C01821=1016.661,-35.852,383.395,-24.107,21.573,-43.343
C01822=1016.661,-36.185,383.421,-24.107,21.574,-43.347
C01823=1016.662,-36.517,383.447,-24.106,21.574,-43.352
C01824=1016.663,-36.850,383.473,-24.105,21.574,-43.357
C01825=1016.662,-37.183,383.498,-24.105,21.575,-43.361
C01826=1016.663,-37.515,383.525,-24.104,21.575,-43.366
C01827=1016.663,-37.848,383.550,-24.103,21.576,-43.371
C01828=1016.663,-38.180,383.576,-24.102,21.576,-43.376
C01829=1016.664,-38.513,383.602,-24.102,21.577,-43.380
C01830=1016.664,-38.846,383.627,-24.101,21.577,-43.385
C01831=1016.665,-39.178,383.654,-24.101,21.578,-43.389
C01832=1016.664,-39.511,383.679,-24.100,21.578,-43.394
C01833=1016.665,-39.844,383.705,-24.100,21.579,-43.398
C01834=1016.664,-40.177,383.731,-24.099,21.579,-43.404
C01835=1016.665,-40.509,383.757,-24.098,21.580,-43.409
C01836=1016.665,-40.842,383.782,-24.098,21.580,-43.413
C01837=1016.665,-41.174,383.808,-24.097,21.580,-43.418
C01838=1016.665,-41.507,383.834,-24.096,21.582,-43.422
C01839=1016.665,-41.839,383.859,-24.096,21.582,-43.427
C01840=1016.666,-42.172,383.885,-24.095,21.582,-43.431
C01841=1016.666,-42.504,383.911,-24.094,21.583,-43.437
C01842=1016.666,-42.837,383.936,-24.094,21.583,-43.442
C01843=1016.665,-43.169,383.962,-24.093,21.583,-43.446
C01844=1016.666,-43.502,383.987,-24.092,21.584,-43.451
C01845=1016.665,-43.835,384.013,-24.092,21.585,-43.455
C01846=1016.665,-44.167,384.039,-24.091,21.585,-43.461
C01847=1016.665,-44.500,384.064,-24.091,21.586,-43.465
C01848=1016.666,-44.833,384.090,-24.090,21.586,-43.470
C01849=1016.666,-45.165,384.116,-24.089,21.586,-43.475
C01850=1016.666,-45.498,384.141,-24.089,21.587,-43.479
C01851=1016.665,-45.830,384.167,-24.088,21.588,-43.485
C01852=1016.665,-46.162,384.192,-24.088,21.588,-43.488
C01853=1016.665,-46.495,384.217,-24.087,21.588,-43.494
C01854=1016.665,-46.827,384.243,-24.086,21.590,-43.498
C01855=1016.664,-47.160,384.269,-24.086,21.589,-43.503
C01856=1016.664,-47.493,384.294,-24.085,21.589,-43.508
C01857=1016.664,-47.825,384.320,-24.084,21.591,-43.512
C01858=1016.664,-48.158,384.345,-24.083,21.591,-43.518
C01859=1016.664,-48.490,384.370,-24.083,21.592,-43.522
C01860=1016.664,-48.822,384.396,-24.082,21.592,-43.527
C01861=1016.664,-49.155,384.421,-24.081,21.592,-43.532
C01862=1016.664,-49.487,384.447,-24.081,21.593,-43.536
C01863=1016.663,-49.820,384.472,-24.080,21.593,-43.542
C01864=1016.663,-50.152,384.497,-24.080,21.595,-43.546
C01865=1016.662,-50.484,384.522,-24.079,21.594,-43.551
C01866=1016.662,-50.817,384.548,-24.079,21.595,-43.555
C01867=1016.662,-51.149,384.573,-24.078,21.596,-43.560
C01868=1016.661,-51.482,384.599,-24.077,21.596,-43.566
C01869=1016.660,-51.814,384.624,-24.077,21.597,-43.570
C01870=1016.661,-52.147,384.649,-24.076,21.597,-43.575
C01871=1016.660,-52.479,384.674,-24.075,21.597,-43.579
C01872=1016.659,-52.811,384.700,-24.075,21.598,-43.584
C01873=1016.659,-53.144,384.725,-24.074,21.598,-43.589
C01874=1016.658,-53.476,384.750,-24.074,21.600,-43.594
C01875=1016.658,-53.808,384.776,-24.073,21.599,-43.599
C01876=1016.658,-54.140,384.800,-24.072,21.600,-43.603
C01877=1016.657,-54.473,384.826,-24.072,21.601,-43.608
C01878=1016.656,-54.805,384.851,-24.071,21.601,-43.613
C01879=1016.656,-55.137,384.876,-24.070,21.602,-43.618
C01880=1016.655,-55.469,384.901,-24.070,21.602,-43.623
C01881=1016.655,-55.803,384.926,-24.069,21.603,-43.627
C01882=1016.655,-56.136,384.951,-24.068,21.603,-43.632
C01883=1016.653,-56.468,384.977,-24.068,21.603,-43.637
C01884=1016.654,-56.801,385.002,-24.067,21.605,-43.642
C01885=1016.653,-57.135,385.027,-24.066,21.604,-43.647
C01886=1016.652,-57.468,385.052,-24.066,21.605,-43.652
C01887=1016.651,-57.803,385.077,-24.065,21.606,-43.656
C01888=1016.650,-58.136,385.102,-24.064,21.606,-43.662
C01889=1016.650,-58.471,385.128,-24.064,21.607,-43.666
C01890=1016.650,-58.806,385.153,-24.063,21.607,-43.671
C01891=1016.649,-59.141,385.178,-24.062,21.608,-43.676
C01892=1016.647,-59.477,385.203,-24.062,21.608,-43.680
C01893=1016.647,-59.813,385.228,-24.061,21.609,-43.686
C01894=1016.646,-60.149,385.254,-24.060,21.609,-43.691
C01895=1016.645,-60.486,385.280,-24.060,21.610,-43.695
C01896=1016.645,-60.823,385.304,-24.059,21.610,-43.700
C01897=1016.644,-61.162,385.330,-24.059,21.611,-43.706
C01898=1016.643,-61.499,385.355,-24.058,21.611,-43.710
C01899=1016.642,-61.838,385.381,-24.057,21.612,-43.715
C01900=1016.641,-62.177,385.406,-24.057,21.612,-43.720
C01901=1016.640,-62.515,385.432,-24.056,21.614,-43.725
C01902=1016.640,-62.855,385.457,-24.055,21.613,-43.730
C01903=1016.638,-63.195,385.482,-24.055,21.614,-43.735
C01904=1016.637,-63.535,385.507,-24.054,21.615,-43.739
C01905=1016.636,-63.876,385.533,-24.053,21.616,-43.745
C01906=1016.636,-64.217,385.558,-24.053,21.615,-43.750
C01907=1016.634,-64.558,385.584,-24.052,21.617,-43.754
C01908=1016.634,-64.900,385.609,-24.051,21.617,-43.759
C01909=1016.632,-65.242,385.635,-24.051,21.618,-43.765
C01910=1016.631,-65.584,385.660,-24.050,21.617,-43.770
C01911=1016.630,-65.926,385.686,-24.050,21.619,-43.774
C01912=1016.629,-66.269,385.711,-24.049,21.619,-43.780
C01913=1016.628,-66.612,385.737,-24.048,21.620,-43.785
C01914=1016.626,-66.955,385.762,-24.048,21.620,-43.789
C01915=1016.626,-67.298,385.787,-24.047,21.621,-43.795
C01916=1016.624,-67.641,385.814,-24.046,21.621,-43.800
C01917=1016.623,-67.984,385.839,-24.045,21.622,-43.805
C01918=1016.621,-68.328,385.864,-24.045,21.622,-43.809
C01919=1016.620,-68.672,385.890,-24.044,21.623,-43.815
C01920=1016.620,-69.016,385.915,-24.043,21.623,-43.820
C01921=1016.619,-69.360,385.941,-24.043,21.624,-43.824
C01922=1016.617,-69.704,385.966,-24.042,21.624,-43.829
C01923=1016.615,-70.047,385.992,-24.041,21.625,-43.835
C01924=1016.614,-70.391,386.017,-24.041,21.625,-43.840
C01925=1016.613,-70.736,386.042,-24.040,21.626,-43.844
C01926=1016.611,-71.080,386.068,-24.040,21.627,-43.850
C01927=1016.610,-71.424,386.093,-24.039,21.627,-43.855
C01928=1016.609,-71.768,386.118,-24.038,21.628,-43.861
C01929=1016.608,-72.112,386.144,-24.038,21.628,-43.865
C01930=1016.606,-72.456,386.169,-24.037,21.629,-43.870
C01931=1016.604,-72.800,386.195,-24.036,21.629,-43.875
C01932=1016.603,-73.144,386.220,-24.035,21.630,-43.881
C01933=1016.602,-73.488,386.245,-24.035,21.630,-43.885
C01934=1016.600,-73.831,386.270,-24.034,21.631,-43.890
C01935=1016.598,-74.175,386.296,-24.033,21.632,-43.896
C01936=1016.596,-74.519,386.321,-24.033,21.632,-43.901
C01937=1016.595,-74.862,386.346,-24.032,21.633,-43.905
C01938=1016.594,-75.206,386.372,-24.031,21.633,-43.911
C01939=1016.592,-75.549,386.397,-24.031,21.634,-43.916
C01940=1016.590,-75.892,386.422,-24.030,21.634,-43.920
C01941=1016.589,-76.235,386.447,-24.030,21.635,-43.926
C01942=1016.587,-76.578,386.472,-24.029,21.635,-43.931
C01943=1016.585,-76.920,386.498,-24.028,21.636,-43.936
C01944=1016.583,-77.263,386.522,-24.028,21.636,-43.940
C01945=1016.582,-77.604,386.547,-24.027,21.637,-43.946
C01946=1016.580,-77.946,386.572,-24.026,21.637,-43.951
C01947=1016.579,-78.288,386.597,-24.026,21.639,-43.955
C01948=1016.577,-78.629,386.622,-24.025,21.638,-43.960
C01949=1016.575,-78.970,386.647,-24.024,21.639,-43.966
C01950=1016.573,-79.310,386.672,-24.023,21.639,-43.971
C01951=1016.571,-79.651,386.697,-24.023,21.641,-43.975
C01952=1016.570,-79.990,386.722,-24.022,21.641,-43.981
C01953=1016.568,-80.329,386.746,-24.021,21.641,-43.986
C01954=1016.566,-80.669,386.770,-24.021,21.643,-43.990
C01955=1016.564,-81.007,386.796,-24.020,21.643,-43.995
C01956=1016.562,-81.345,386.820,-24.020,21.643,-44.001
C01957=1016.560,-81.683,386.844,-24.019,21.644,-44.005
C01958=1016.558,-82.020,386.869,-24.018,21.645,-44.010
C01959=1016.556,-82.358,386.894,-24.018,21.645,-44.016
C01960=1016.555,-82.694,386.918,-24.017,21.645,-44.021
C01961=1016.552,-83.030,386.942,-24.016,21.646,-44.025
C01962=1016.550,-83.366,386.967,-24.016,21.647,-44.031
C01963=1016.549,-83.701,386.991,-24.015,21.647,-44.036
C01964=1016.547,-84.036,387.015,-24.015,21.648,-44.040
C01965=1016.544,-84.370,387.039,-24.014,21.648,-44.045
C01966=1016.542,-84.719,387.065,-24.013,21.649,-44.051
C01967=1016.540,-85.117,387.094,-24.012,21.650,-44.056
C01968=1016.538,-85.330,387.109,-24.012,21.649,-44.060
C01969=1016.538,-85.543,387.124,-24.012,21.649,-44.062
C01970=1016.535,-85.951,387.154,-24.011,21.650,-44.067
C01971=1016.532,-86.311,387.179,-24.010,21.651,-44.073
C01972=1016.531,-86.640,387.203,-24.009,21.652,-44.078
C01973=1016.528,-86.963,387.226,-24.009,21.652,-44.082
C01974=1016.526,-87.279,387.250,-24.008,21.653,-44.088
C01975=1016.524,-87.591,387.272,-24.007,21.653,-44.093
C01976=1016.522,-87.902,387.294,-24.007,21.654,-44.097
C01977=1016.520,-88.215,387.317,-24.006,21.654,-44.102
C01978=1016.518,-88.533,387.340,-24.006,21.655,-44.106
C01979=1016.515,-88.905,387.367,-24.005,21.656,-44.114
C01980=1016.514,-89.123,387.382,-24.004,21.656,-44.117
C01981=1016.512,-89.358,387.399,-24.004,21.656,-44.119
C01982=1016.510,-89.596,387.416,-24.004,21.656,-44.121
C01983=1016.509,-89.827,387.433,-24.004,21.657,-44.123
C01984=1016.506,-90.233,387.462,-24.003,21.658,-44.130
C01985=1016.503,-90.571,387.486,-24.002,21.658,-44.136
C01986=1016.502,-90.901,387.510,-24.001,21.659,-44.141
C01987=1016.499,-91.230,387.533,-24.001,21.660,-44.145
C01988=1016.496,-91.558,387.557,-24.000,21.660,-44.150
C01989=1016.494,-91.887,387.580,-23.999,21.660,-44.156
C01990=1016.492,-92.215,387.604,-23.999,21.661,-44.160
C01991=1016.489,-92.542,387.627,-23.998,21.662,-44.165
C01992=1016.487,-92.868,387.651,-23.998,21.662,-44.169
C01993=1016.484,-93.195,387.673,-23.997,21.663,-44.175
C01994=1016.482,-93.520,387.697,-23.996,21.663,-44.180
C01995=1016.479,-93.846,387.721,-23.996,21.664,-44.184
C01996=1016.477,-94.171,387.743,-23.995,21.664,-44.189
C01997=1016.474,-94.494,387.766,-23.994,21.665,-44.193
C01998=1016.471,-94.818,387.790,-23.994,21.666,-44.199
C01999=1016.469,-95.140,387.812,-23.993,21.666,-44.204
C02000=1016.467,-95.463,387.836,-23.993,21.666,-44.207
C02001=1016.465,-95.786,387.859,-23.992,21.667,-44.213
C02002=1016.461,-96.108,387.882,-23.991,21.668,-44.217
C02003=1016.459,-96.429,387.904,-23.991,21.668,-44.222
C02004=1016.456,-96.751,387.927,-23.990,21.669,-44.226
C02005=1016.453,-97.072,387.950,-23.989,21.669,-44.231
C02006=1016.451,-97.393,387.973,-23.989,21.670,-44.236
C02007=1016.449,-97.713,387.995,-23.988,21.670,-44.241
C02008=1016.446,-98.035,388.019,-23.987,21.670,-44.246
C02009=1016.443,-98.356,388.041,-23.987,21.672,-44.250
C02010=1016.441,-98.676,388.064,-23.986,21.671,-44.255
C02011=1016.438,-98.998,388.087,-23.986,21.673,-44.260
C02012=1016.436,-99.319,388.109,-23.985,21.673,-44.265
C02013=1016.432,-99.640,388.132,-23.985,21.673,-44.268
C02014=1016.429,-99.962,388.154,-23.984,21.674,-44.274
C02015=1016.427,-100.284,388.177,-23.983,21.675,-44.278
C02016=1016.424,-100.606,388.200,-23.983,21.675,-44.283
C02017=1016.421,-100.928,388.223,-23.982,21.676,-44.287
C02018=1016.419,-101.252,388.246,-23.981,21.676,-44.292
C02019=1016.415,-101.575,388.269,-23.981,21.677,-44.298
C02020=1016.412,-101.899,388.292,-23.980,21.677,-44.302
C02021=1016.409,-102.224,388.315,-23.980,21.678,-44.307
C02022=1016.407,-102.549,388.337,-23.979,21.679,-44.311
C02023=1016.403,-102.874,388.360,-23.978,21.679,-44.316
C02024=1016.400,-103.201,388.384,-23.978,21.680,-44.320
C02025=1016.397,-103.527,388.406,-23.977,21.680,-44.326
C02026=1016.395,-103.854,388.429,-23.976,21.681,-44.331
C02027=1016.392,-104.181,388.452,-23.976,21.681,-44.335
C02028=1016.388,-104.509,388.475,-23.975,21.681,-44.340
C02029=1016.385,-104.837,388.498,-23.975,21.683,-44.344
C02030=1016.381,-105.165,388.521,-23.974,21.683,-44.350
C02031=1016.379,-105.494,388.545,-23.974,21.684,-44.354
C02032=1016.376,-105.823,388.567,-23.973,21.684,-44.359
C02033=1016.372,-106.151,388.591,-23.972,21.685,-44.365
C02034=1016.369,-106.480,388.614,-23.972,21.685,-44.368
C02035=1016.365,-106.809,388.637,-23.971,21.685,-44.374
C02036=1016.363,-107.139,388.661,-23.971,21.687,-44.378
C02037=1016.359,-107.467,388.683,-23.970,21.687,-44.383
C02038=1016.356,-107.797,388.706,-23.969,21.687,-44.388
C02039=1016.353,-108.125,388.729,-23.969,21.688,-44.392
C02040=1016.349,-108.455,388.752,-23.968,21.689,-44.398
C02041=1016.346,-108.784,388.775,-23.967,21.689,-44.402
C02042=1016.343,-109.112,388.798,-23.967,21.689,-44.407
C02043=1016.339,-109.442,388.821,-23.966,21.690,-44.412
C02044=1016.336,-109.770,388.844,-23.965,21.691,-44.416
C02045=1016.332,-110.100,388.867,-23.965,21.691,-44.422
C02046=1016.329,-110.428,388.889,-23.964,21.692,-44.426
C02047=1016.325,-110.757,388.913,-23.963,21.692,-44.431
C02048=1016.322,-111.086,388.936,-23.963,21.693,-44.436
C02049=1016.318,-111.414,388.958,-23.962,21.693,-44.440
C02050=1016.314,-111.744,388.981,-23.962,21.694,-44.446
C02051=1016.311,-112.072,389.004,-23.961,21.695,-44.449
C02052=1016.308,-112.401,389.027,-23.960,21.695,-44.455
C02053=1016.304,-112.730,389.050,-23.960,21.696,-44.459
C02054=1016.300,-113.058,389.073,-23.959,21.696,-44.464
C02055=1016.297,-113.387,389.096,-23.958,21.697,-44.470
C02056=1016.293,-113.716,389.119,-23.958,21.697,-44.473
C02057=1016.289,-114.044,389.141,-23.957,21.698,-44.479
C02058=1016.285,-114.373,389.165,-23.957,21.699,-44.483
C02059=1016.282,-114.701,389.187,-23.956,21.699,-44.488
C02060=1016.278,-115.031,389.210,-23.956,21.700,-44.492
C02061=1016.274,-115.359,389.232,-23.955,21.700,-44.497
C02062=1016.270,-115.688,389.256,-23.954,21.701,-44.503
C02063=1016.267,-116.016,389.278,-23.954,21.701,-44.507
C02064=1016.263,-116.345,389.301,-23.953,21.701,-44.512
C02065=1016.259,-116.673,389.324,-23.953,21.703,-44.516
C02066=1016.255,-117.001,389.346,-23.952,21.703,-44.521
C02067=1016.251,-117.330,389.369,-23.951,21.704,-44.525
C02068=1016.248,-117.659,389.391,-23.951,21.704,-44.531
C02069=1016.243,-117.987,389.414,-23.950,21.705,-44.535
C02070=1016.240,-118.315,389.437,-23.949,21.705,-44.540
C02071=1016.236,-118.644,389.459,-23.949,21.705,-44.545
C02072=1016.231,-118.972,389.482,-23.948,21.707,-44.549
C02073=1016.227,-119.301,389.505,-23.948,21.707,-44.554
C02074=1016.224,-119.629,389.528,-23.947,21.707,-44.558
C02075=1016.219,-119.958,389.550,-23.946,21.708,-44.564
C02076=1016.216,-120.286,389.573,-23.946,21.709,-44.568
C02077=1016.212,-120.614,389.595,-23.945,21.709,-44.573
C02078=1016.207,-120.943,389.618,-23.945,21.710,-44.577
C02079=1016.203,-121.270,389.641,-23.944,21.710,-44.582
C02080=1016.199,-121.599,389.663,-23.944,21.711,-44.586
C02081=1016.195,-121.928,389.685,-23.943,21.711,-44.591
C02082=1016.190,-122.256,389.708,-23.942,21.712,-44.597
C02083=1016.186,-122.584,389.730,-23.942,21.713,-44.601
C02084=1016.182,-122.913,389.754,-23.941,21.713,-44.606
C02085=1016.178,-123.241,389.776,-23.940,21.714,-44.610
C02086=1016.173,-123.569,389.799,-23.940,21.714,-44.615
C02087=1016.169,-123.897,389.820,-23.939,21.715,-44.620
C02088=1016.165,-124.225,389.843,-23.939,21.715,-44.625
C02089=1016.160,-124.554,389.866,-23.938,21.716,-44.628
C02090=1016.157,-124.882,389.888,-23.937,21.717,-44.634
C02091=1016.152,-125.210,389.911,-23.937,21.717,-44.638
C02092=1016.147,-125.538,389.933,-23.936,21.717,-44.643
C02093=1016.143,-125.867,389.956,-23.936,21.719,-44.647
C02094=1016.139,-126.195,389.978,-23.935,21.719,-44.652
C02095=1016.134,-126.523,390.000,-23.935,21.720,-44.657
C02096=1016.129,-126.850,390.023,-23.934,21.720,-44.662
C02097=1016.125,-127.179,390.046,-23.933,21.720,-44.667
C02098=1016.120,-127.507,390.068,-23.933,21.721,-44.671
C02099=1016.116,-127.836,390.090,-23.932,21.721,-44.676
C02100=1016.111,-128.163,390.113,-23.931,21.722,-44.680
C02101=1016.107,-128.492,390.135,-23.931,21.723,-44.686
C02102=1016.102,-128.819,390.157,-23.930,21.723,-44.689
C02103=1016.097,-129.148,390.180,-23.929,21.723,-44.695
C02104=1016.093,-129.476,390.202,-23.929,21.725,-44.699
C02105=1016.088,-129.804,390.224,-23.928,21.724,-44.704
C02106=1016.083,-130.132,390.247,-23.928,21.726,-44.708
C02107=1016.078,-130.460,390.269,-23.927,21.726,-44.713
C02108=1016.074,-130.789,390.292,-23.927,21.726,-44.717
C02109=1016.069,-131.116,390.314,-23.926,21.727,-44.723
C02110=1016.064,-131.445,390.336,-23.926,21.728,-44.726
C02111=1016.059,-131.772,390.358,-23.925,21.728,-44.732
C02112=1016.054,-132.100,390.381,-23.924,21.729,-44.736
C02113=1016.050,-132.428,390.403,-23.924,21.729,-44.741
C02114=1016.044,-132.756,390.425,-23.923,21.730,-44.745
C02115=1016.039,-133.085,390.447,-23.922,21.731,-44.750
C02116=1016.034,-133.412,390.469,-23.922,21.731,-44.754
C02117=1016.029,-133.740,390.492,-23.921,21.731,-44.759
C02118=1016.025,-134.069,390.514,-23.921,21.732,-44.763
C02119=1016.426,-134.039,390.264,-23.921,21.732,-44.763
C02120=1016.431,-133.712,390.241,-23.921,21.731,-44.759
C02121=1016.436,-133.383,390.220,-23.922,21.731,-44.754
C02122=1016.441,-133.056,390.197,-23.922,21.731,-44.750
C02123=1016.446,-132.727,390.175,-23.923,21.730,-44.745
C02124=1016.450,-132.400,390.153,-23.924,21.729,-44.741
C02125=1016.455,-132.072,390.131,-23.924,21.729,-44.736
C02126=1016.460,-131.744,390.109,-23.925,21.728,-44.732
C02127=1016.464,-131.415,390.086,-23.926,21.728,-44.726
C02128=1016.469,-131.087,390.064,-23.926,21.727,-44.723
C02129=1016.474,-130.759,390.042,-23.927,21.726,-44.717
C02130=1016.477,-130.431,390.020,-23.927,21.726,-44.713
C02131=1016.483,-130.103,389.998,-23.928,21.726,-44.708
C02132=1016.487,-129.775,389.976,-23.928,21.724,-44.704
C02133=1016.492,-129.447,389.953,-23.929,21.725,-44.699
C02134=1016.496,-129.119,389.931,-23.929,21.723,-44.695
C02135=1016.501,-128.791,389.909,-23.930,21.723,-44.689
C02136=1016.505,-128.462,389.886,-23.931,21.723,-44.686
C02137=1016.510,-128.135,389.864,-23.931,21.722,-44.680
C02138=1016.514,-127.807,389.842,-23.932,21.721,-44.676
C02139=1016.519,-127.478,389.820,-23.933,21.721,-44.671
C02140=1016.523,-127.150,389.797,-23.933,21.720,-44.667
C02141=1016.527,-126.822,389.775,-23.934,21.720,-44.662
C02142=1016.532,-126.494,389.752,-23.935,21.720,-44.657
C02143=1016.536,-126.166,389.730,-23.935,21.719,-44.652
C02144=1016.540,-125.837,389.708,-23.936,21.719,-44.647
C02145=1016.545,-125.510,389.686,-23.936,21.717,-44.643
C02146=1016.549,-125.181,389.664,-23.937,21.717,-44.638
C02147=1016.553,-124.853,389.640,-23.937,21.717,-44.634
C02148=1016.557,-124.525,389.618,-23.938,21.716,-44.628
C02149=1016.561,-124.197,389.596,-23.939,21.715,-44.625
C02150=1016.566,-123.868,389.573,-23.939,21.715,-44.620
C02151=1016.569,-123.540,389.551,-23.940,21.714,-44.615
C02152=1016.574,-123.212,389.529,-23.940,21.714,-44.610
C02153=1016.579,-122.884,389.506,-23.941,21.713,-44.606
C02154=1016.582,-122.555,389.484,-23.942,21.713,-44.601
C02155=1016.586,-122.227,389.462,-23.942,21.712,-44.597
C02156=1016.591,-121.899,389.439,-23.943,21.711,-44.591
C02157=1016.595,-121.571,389.417,-23.944,21.711,-44.586
C02158=1016.598,-121.242,389.395,-23.944,21.710,-44.582
C02159=1016.602,-120.914,389.371,-23.945,21.710,-44.577
C02160=1016.606,-120.585,389.349,-23.945,21.709,-44.573
C02161=1016.610,-120.257,389.327,-23.946,21.709,-44.568
C02162=1016.615,-119.929,389.303,-23.946,21.708,-44.564
C02163=1016.618,-119.601,389.281,-23.947,21.707,-44.558
C02164=1016.622,-119.272,389.259,-23.948,21.707,-44.554
C02165=1016.626,-118.943,389.236,-23.948,21.707,-44.549
C02166=1016.630,-118.615,389.213,-23.949,21.705,-44.545
C02167=1016.634,-118.287,389.191,-23.949,21.705,-44.540
C02168=1016.638,-117.958,389.169,-23.950,21.705,-44.535
C02169=1016.641,-117.630,389.146,-23.951,21.704,-44.531
C02170=1016.645,-117.302,389.123,-23.951,21.704,-44.525
C02171=1016.649,-116.973,389.100,-23.952,21.703,-44.521
C02172=1016.652,-116.644,389.078,-23.953,21.703,-44.516
C02173=1016.656,-116.316,389.056,-23.953,21.701,-44.512
C02174=1016.660,-115.987,389.033,-23.954,21.701,-44.507
C02175=1016.664,-115.659,389.010,-23.954,21.701,-44.503
C02176=1016.667,-115.331,388.987,-23.955,21.700,-44.497
C02177=1016.671,-115.001,388.964,-23.956,21.700,-44.492
C02178=1016.674,-114.673,388.942,-23.956,21.699,-44.488
C02179=1016.677,-114.345,388.920,-23.957,21.699,-44.483
C02180=1016.682,-114.016,388.896,-23.957,21.698,-44.479
C02181=1016.685,-113.688,388.874,-23.958,21.697,-44.473
C02182=1016.689,-113.358,388.851,-23.958,21.697,-44.470
C02183=1016.693,-113.030,388.829,-23.959,21.696,-44.464
C02184=1016.696,-112.702,388.806,-23.960,21.696,-44.459
C02185=1016.699,-112.372,388.783,-23.960,21.695,-44.455
C02186=1016.702,-112.044,388.760,-23.961,21.695,-44.449
C02187=1016.707,-111.715,388.738,-23.962,21.694,-44.446
C02188=1016.710,-111.386,388.715,-23.962,21.693,-44.440
C02189=1016.713,-111.058,388.692,-23.963,21.693,-44.436
C02190=1016.717,-110.729,388.668,-23.963,21.692,-44.431
C02191=1016.720,-110.400,388.646,-23.964,21.692,-44.426
C02192=1016.723,-110.071,388.623,-23.965,21.691,-44.422
C02193=1016.726,-109.743,388.600,-23.965,21.691,-44.416
C02194=1016.730,-109.413,388.577,-23.966,21.690,-44.412
C02195=1016.733,-109.085,388.554,-23.967,21.689,-44.407
C02196=1016.737,-108.755,388.531,-23.967,21.689,-44.402
C02197=1016.740,-108.427,388.508,-23.968,21.689,-44.398
C02198=1016.743,-108.098,388.485,-23.969,21.688,-44.392
C02199=1016.746,-107.769,388.463,-23.969,21.687,-44.388
C02200=1016.749,-107.439,388.439,-23.970,21.687,-44.383
C02201=1016.752,-107.110,388.417,-23.971,21.687,-44.378
C02202=1016.756,-106.781,388.394,-23.971,21.685,-44.374
C02203=1016.759,-106.452,388.371,-23.972,21.685,-44.368
C02204=1016.762,-106.123,388.348,-23.972,21.685,-44.365
C02205=1016.765,-105.794,388.325,-23.973,21.684,-44.359
C02206=1016.768,-105.466,388.302,-23.974,21.684,-44.354
C02207=1016.771,-105.138,388.279,-23.974,21.683,-44.350
C02208=1016.774,-104.809,388.256,-23.975,21.683,-44.344
C02209=1016.777,-104.481,388.233,-23.975,21.681,-44.340
C02210=1016.780,-104.153,388.210,-23.976,21.681,-44.335
C02211=1016.783,-103.825,388.187,-23.976,21.681,-44.331
C02212=1016.786,-103.499,388.163,-23.977,21.680,-44.326
C02213=1016.789,-103.173,388.141,-23.978,21.680,-44.320
C02214=1016.791,-102.847,388.118,-23.978,21.679,-44.316
C02215=1016.795,-102.521,388.095,-23.979,21.679,-44.311
C02216=1016.798,-102.196,388.072,-23.980,21.678,-44.307
C02217=1016.800,-101.871,388.050,-23.980,21.677,-44.302
C02218=1016.803,-101.546,388.027,-23.981,21.677,-44.298
C02219=1016.806,-101.223,388.004,-23.981,21.676,-44.292
C02220=1016.809,-100.900,387.981,-23.982,21.676,-44.287
C02221=1016.812,-100.577,387.959,-23.983,21.675,-44.283
C02222=1016.815,-100.255,387.936,-23.983,21.675,-44.278
C02223=1016.817,-99.933,387.913,-23.984,21.674,-44.274
C02224=1016.820,-99.612,387.890,-23.985,21.673,-44.268
C02225=1016.822,-99.291,387.868,-23.985,21.673,-44.265
C02226=1016.826,-98.970,387.845,-23.986,21.673,-44.260
C02227=1016.828,-98.649,387.823,-23.986,21.671,-44.255
C02228=1016.831,-98.327,387.800,-23.987,21.672,-44.250
C02229=1016.833,-98.007,387.777,-23.987,21.670,-44.246
C02230=1016.836,-97.686,387.755,-23.988,21.670,-44.241
C02231=1016.838,-97.365,387.732,-23.989,21.670,-44.236
C02232=1016.841,-97.044,387.708,-23.989,21.669,-44.231
C02233=1016.843,-96.723,387.686,-23.990,21.669,-44.226
C02234=1016.846,-96.402,387.663,-23.991,21.668,-44.222
C02235=1016.849,-96.080,387.640,-23.991,21.668,-44.217
C02236=1016.851,-95.757,387.617,-23.992,21.667,-44.213
C02237=1016.854,-95.436,387.595,-23.993,21.666,-44.207
C02238=1016.856,-95.113,387.572,-23.993,21.666,-44.204
C02239=1016.858,-94.790,387.549,-23.994,21.666,-44.199
C02240=1016.861,-94.466,387.526,-23.994,21.665,-44.193
C02241=1016.863,-94.142,387.503,-23.995,21.664,-44.189
C02242=1016.866,-93.818,387.479,-23.996,21.664,-44.184
C02243=1016.868,-93.493,387.457,-23.996,21.663,-44.180
C02244=1016.871,-93.167,387.433,-23.997,21.663,-44.175
C02245=1016.873,-92.841,387.410,-23.998,21.662,-44.169
C02246=1016.875,-92.513,387.386,-23.998,21.662,-44.165
C02247=1016.878,-92.186,387.363,-23.999,21.661,-44.160
C02248=1016.880,-91.859,387.340,-23.999,21.660,-44.156
C02249=1016.882,-91.530,387.316,-24.000,21.660,-44.150
C02250=1016.885,-91.201,387.292,-24.001,21.660,-44.145
C02251=1016.887,-90.873,387.269,-24.001,21.659,-44.141
C02252=1016.889,-90.543,387.246,-24.002,21.658,-44.136
C02253=1016.891,-90.205,387.222,-24.003,21.658,-44.130
C02254=1016.894,-89.799,387.193,-24.004,21.657,-44.123
C02255=1016.896,-89.568,387.176,-24.004,21.656,-44.121
C02256=1016.898,-89.330,387.159,-24.004,21.656,-44.119
C02257=1016.899,-89.096,387.142,-24.004,21.656,-44.117
C02258=1016.901,-88.877,387.126,-24.005,21.656,-44.114
C02259=1016.903,-88.506,387.100,-24.006,21.655,-44.106
C02260=1016.905,-88.187,387.077,-24.006,21.654,-44.102
C02261=1016.907,-87.874,387.054,-24.007,21.654,-44.097
C02262=1016.908,-87.564,387.032,-24.007,21.653,-44.093
C02263=1016.911,-87.251,387.009,-24.008,21.653,-44.088
C02264=1016.913,-86.935,386.987,-24.009,21.652,-44.082
C02265=1016.915,-86.612,386.964,-24.009,21.652,-44.078
C02266=1016.917,-86.283,386.940,-24.010,21.651,-44.073
C02267=1016.919,-85.924,386.914,-24.011,21.650,-44.067
C02268=1016.921,-85.515,386.884,-24.012,21.649,-44.062
C02269=1016.923,-85.301,386.869,-24.012,21.649,-44.060
C02270=1016.924,-85.089,386.853,-24.012,21.650,-44.056
C02271=1016.927,-84.692,386.825,-24.013,21.649,-44.051
C02272=1016.929,-84.342,386.800,-24.014,21.648,-44.045
C02273=1016.930,-84.008,386.775,-24.015,21.648,-44.040
C02274=1016.933,-83.674,386.752,-24.015,21.647,-44.036
C02275=1016.935,-83.338,386.728,-24.016,21.647,-44.031
C02276=1016.937,-83.002,386.703,-24.016,21.646,-44.025
C02277=1016.939,-82.667,386.679,-24.017,21.645,-44.021
C02278=1016.940,-82.330,386.654,-24.018,21.645,-44.016
C02279=1016.942,-81.992,386.630,-24.018,21.645,-44.010
C02280=1016.944,-81.655,386.605,-24.019,21.644,-44.005
C02281=1016.946,-81.317,386.580,-24.020,21.643,-44.001
C02282=1016.947,-80.980,386.556,-24.020,21.643,-43.995
C02283=1016.949,-80.641,386.532,-24.021,21.643,-43.990
C02284=1016.952,-80.302,386.507,-24.021,21.641,-43.986
C02285=1016.953,-79.962,386.482,-24.022,21.641,-43.981
C02286=1016.955,-79.622,386.457,-24.023,21.641,-43.975
C02287=1016.956,-79.282,386.432,-24.023,21.639,-43.971
C02288=1016.958,-78.942,386.407,-24.024,21.639,-43.966
C02289=1016.960,-78.601,386.383,-24.025,21.638,-43.960
C02290=1016.962,-78.260,386.358,-24.026,21.639,-43.955
C02291=1016.963,-77.918,386.334,-24.026,21.637,-43.951
C02292=1016.965,-77.576,386.308,-24.027,21.637,-43.946
C02293=1016.967,-77.235,386.284,-24.028,21.636,-43.940
C02294=1016.969,-76.892,386.258,-24.028,21.636,-43.936
C02295=1016.970,-76.550,386.233,-24.029,21.635,-43.931
C02296=1016.972,-76.207,386.208,-24.030,21.635,-43.926
C02297=1016.973,-75.800,386.179,-24.030,21.634,-43.920
C02298=1016.975,-75.521,386.158,-24.031,21.634,-43.916
C02299=1016.977,-75.178,386.133,-24.031,21.633,-43.911
C02300=1016.978,-74.835,386.108,-24.032,21.633,-43.905
C02301=1016.979,-74.491,386.083,-24.033,21.632,-43.901
C02302=1016.981,-74.147,386.057,-24.033,21.632,-43.896
C02303=1016.982,-73.804,386.032,-24.034,21.631,-43.890
C02304=1016.984,-73.460,386.007,-24.035,21.630,-43.885
C02305=1016.985,-73.116,385.981,-24.035,21.630,-43.881
C02306=1016.987,-72.772,385.957,-24.036,21.629,-43.875
C02307=1016.988,-72.428,385.931,-24.037,21.629,-43.870
C02308=1016.990,-72.085,385.906,-24.038,21.628,-43.865
C02309=1016.991,-71.740,385.881,-24.038,21.628,-43.861
C02310=1016.992,-71.396,385.855,-24.039,21.627,-43.855
C02311=1016.993,-71.052,385.829,-24.040,21.627,-43.850
C02312=1016.995,-70.708,385.805,-24.040,21.626,-43.844
C02313=1016.996,-70.364,385.779,-24.041,21.625,-43.840
C02314=1016.998,-70.020,385.753,-24.041,21.625,-43.835
C02315=1016.999,-69.676,385.727,-24.042,21.624,-43.829
C02316=1017.001,-69.332,385.703,-24.043,21.624,-43.824
C02317=1017.002,-68.988,385.677,-24.043,21.623,-43.820
C02318=1017.002,-68.645,385.652,-24.044,21.623,-43.815
C02319=1017.004,-68.301,385.626,-24.045,21.622,-43.809
C02320=1017.005,-67.957,385.600,-24.045,21.622,-43.805
C02321=1017.006,-67.614,385.575,-24.046,21.621,-43.800
C02322=1017.008,-67.270,385.550,-24.047,21.621,-43.795
C02323=1017.008,-66.927,385.524,-24.048,21.620,-43.789
C02324=1017.010,-66.584,385.499,-24.048,21.620,-43.785
C02325=1017.011,-66.241,385.473,-24.049,21.619,-43.780
C02326=1017.012,-65.899,385.448,-24.050,21.619,-43.774
C02327=1017.012,-65.556,385.423,-24.050,21.617,-43.770
C02328=1017.014,-65.214,385.397,-24.051,21.618,-43.765
C02329=1017.014,-64.872,385.371,-24.051,21.617,-43.759
C02330=1017.015,-64.531,385.346,-24.052,21.617,-43.754
C02331=1017.017,-64.190,385.320,-24.053,21.615,-43.750
C02332=1017.018,-63.848,385.295,-24.053,21.616,-43.745
C02333=1017.019,-63.508,385.270,-24.054,21.615,-43.739
C02334=1017.020,-63.168,385.244,-24.055,21.614,-43.735
C02335=1017.020,-62.827,385.219,-24.055,21.613,-43.730
C02336=1017.022,-62.489,385.193,-24.056,21.614,-43.725
C02337=1017.022,-62.149,385.168,-24.057,21.612,-43.720
C02338=1017.024,-61.810,385.143,-24.057,21.612,-43.715
C02339=1017.024,-61.472,385.117,-24.058,21.611,-43.710
C02340=1017.025,-61.133,385.092,-24.059,21.611,-43.706
C02341=1017.026,-60.796,385.066,-24.059,21.610,-43.700
C02342=1017.026,-60.458,385.041,-24.060,21.610,-43.695
C02343=1017.027,-60.122,385.016,-24.060,21.609,-43.691
C02344=1017.028,-59.786,384.991,-24.061,21.609,-43.686
C02345=1017.029,-59.449,384.966,-24.062,21.608,-43.680
C02346=1017.030,-59.114,384.940,-24.062,21.608,-43.676
C02347=1017.030,-58.779,384.915,-24.063,21.607,-43.671
C02348=1017.031,-58.444,384.890,-24.064,21.607,-43.666
C02349=1017.032,-58.109,384.865,-24.064,21.606,-43.662
C02350=1017.032,-57.775,384.840,-24.065,21.606,-43.656
C02351=1017.033,-57.440,384.814,-24.066,21.605,-43.652
C02352=1017.034,-57.107,384.789,-24.066,21.604,-43.647
C02353=1017.035,-56.774,384.764,-24.067,21.605,-43.642
C02354=1017.035,-56.441,384.739,-24.068,21.603,-43.637
C02355=1017.035,-56.107,384.714,-24.068,21.603,-43.632
C02356=1017.036,-55.775,384.689,-24.069,21.603,-43.627
C02357=1017.037,-55.442,384.664,-24.070,21.602,-43.623
C02358=1017.037,-55.110,384.638,-24.070,21.602,-43.618
C02359=1017.038,-54.777,384.613,-24.071,21.601,-43.613
C02360=1017.038,-54.445,384.588,-24.072,21.601,-43.608
C02361=1017.039,-54.113,384.563,-24.072,21.600,-43.603
C02362=1017.039,-53.780,384.538,-24.073,21.599,-43.599
C02363=1017.040,-53.448,384.513,-24.074,21.600,-43.594
C02364=1017.040,-53.116,384.488,-24.074,21.598,-43.589
C02365=1017.040,-52.783,384.462,-24.075,21.598,-43.584
C02366=1017.041,-52.452,384.437,-24.075,21.597,-43.579
C02367=1017.041,-52.119,384.412,-24.076,21.597,-43.575
C02368=1017.042,-51.787,384.387,-24.077,21.597,-43.570
C02369=1017.042,-51.455,384.361,-24.077,21.596,-43.566
C02370=1017.042,-51.122,384.336,-24.078,21.596,-43.560
C02371=1017.042,-50.790,384.310,-24.079,21.595,-43.555
C02372=1017.043,-50.458,384.285,-24.079,21.594,-43.551
C02373=1017.043,-50.125,384.260,-24.080,21.595,-43.546
C02374=1017.043,-49.793,384.235,-24.080,21.593,-43.542
C02375=1017.044,-49.460,384.209,-24.081,21.593,-43.536
C02376=1017.044,-49.127,384.184,-24.081,21.592,-43.532
C02377=1017.044,-48.795,384.158,-24.082,21.592,-43.527
C02378=1017.044,-48.462,384.133,-24.083,21.592,-43.522
C02379=1017.045,-48.130,384.108,-24.083,21.591,-43.518
C02380=1017.045,-47.798,384.082,-24.084,21.591,-43.512
C02381=1017.045,-47.465,384.057,-24.085,21.589,-43.508
C02382=1017.046,-47.133,384.032,-24.086,21.589,-43.503
C02383=1017.046,-46.801,384.006,-24.086,21.590,-43.498
C02384=1017.045,-46.467,383.980,-24.087,21.588,-43.494
C02385=1017.045,-46.135,383.955,-24.088,21.588,-43.488
C02386=1017.045,-45.802,383.930,-24.088,21.588,-43.485
C02387=1017.045,-45.470,383.904,-24.089,21.587,-43.479
C02388=1017.046,-45.137,383.878,-24.089,21.586,-43.475
C02389=1017.046,-44.805,383.853,-24.090,21.586,-43.470
C02390=1017.046,-44.472,383.827,-24.091,21.586,-43.465
C02391=1017.047,-44.140,383.802,-24.091,21.585,-43.461
C02392=1017.046,-43.807,383.776,-24.092,21.585,-43.455
C02393=1017.046,-43.475,383.750,-24.092,21.584,-43.451
C02394=1017.046,-43.143,383.725,-24.093,21.583,-43.446
C02395=1017.046,-42.810,383.700,-24.094,21.583,-43.442
C02396=1017.046,-42.477,383.673,-24.094,21.583,-43.437
C02397=1017.046,-42.144,383.648,-24.095,21.582,-43.431
C02398=1017.046,-41.812,383.623,-24.096,21.582,-43.427
C02399=1017.046,-41.479,383.596,-24.096,21.582,-43.422
C02400=1017.046,-41.146,383.571,-24.097,21.580,-43.418
C02401=1017.045,-40.814,383.545,-24.098,21.580,-43.413
C02402=1017.045,-40.481,383.519,-24.098,21.580,-43.409
C02403=1017.045,-40.149,383.494,-24.099,21.579,-43.404
C02404=1017.045,-39.816,383.468,-24.100,21.579,-43.398
C02405=1017.045,-39.484,383.442,-24.100,21.578,-43.394
C02406=1017.044,-39.151,383.417,-24.101,21.578,-43.389
C02407=1017.045,-38.819,383.391,-24.101,21.577,-43.385
C02408=1017.044,-38.486,383.365,-24.102,21.577,-43.380
C02409=1017.043,-38.153,383.339,-24.102,21.576,-43.376
C02410=1017.044,-37.820,383.313,-24.103,21.576,-43.371
C02411=1017.044,-37.487,383.287,-24.104,21.575,-43.366
C02412=1017.043,-37.155,383.262,-24.105,21.575,-43.361
C02413=1017.043,-36.822,383.235,-24.105,21.574,-43.357
C02414=1017.042,-36.490,383.209,-24.106,21.574,-43.352
C02415=1017.042,-36.157,383.184,-24.107,21.574,-43.347
C02416=1017.042,-35.824,383.158,-24.107,21.573,-43.343
C02417=1017.041,-35.492,383.132,-24.108,21.573,-43.337
C02418=1017.040,-35.159,383.106,-24.108,21.572,-43.334
C02419=1017.041,-34.826,383.080,-24.109,21.572,-43.328
C02420=1017.040,-34.494,383.054,-24.109,21.571,-43.324
C02421=1017.039,-34.161,383.028,-24.110,21.571,-43.319
C02422=1017.039,-33.828,383.002,-24.111,21.570,-43.315
C02423=1017.038,-33.496,382.976,-24.111,21.570,-43.310
C02424=1017.038,-33.163,382.949,-24.112,21.569,-43.306
C02425=1017.038,-32.830,382.924,-24.113,21.569,-43.301
C02426=1017.038,-32.497,382.898,-24.113,21.568,-43.296
C02427=1017.037,-32.165,382.872,-24.114,21.568,-43.291
C02428=1017.037,-31.832,382.846,-24.114,21.567,-43.287
C02429=1017.036,-31.499,382.820,-24.115,21.567,-43.282
C02430=1017.036,-31.166,382.794,-24.116,21.566,-43.278
C02431=1017.035,-30.834,382.767,-24.116,21.566,-43.273
C02432=1017.034,-30.501,382.742,-24.117,21.565,-43.269
C02433=1017.034,-30.168,382.715,-24.118,21.565,-43.264
C02434=1017.033,-29.836,382.689,-24.118,21.565,-43.260
C02435=1017.032,-29.503,382.664,-24.119,21.564,-43.254
C02436=1017.032,-29.170,382.637,-24.119,21.563,-43.250
C02437=1017.031,-28.837,382.610,-24.120,21.563,-43.245
C02438=1017.030,-28.505,382.584,-24.120,21.562,-43.241
C02439=1017.029,-28.172,382.559,-24.121,21.562,-43.236
C02440=1017.029,-27.839,382.532,-24.122,21.562,-43.232
C02441=1017.028,-27.507,382.506,-24.123,21.562,-43.227
C02442=1017.027,-27.174,382.479,-24.123,21.560,-43.223
C02443=1017.026,-26.841,382.454,-24.124,21.560,-43.217
C02444=1017.026,-26.508,382.427,-24.124,21.560,-43.214
C02445=1017.025,-26.176,382.401,-24.125,21.559,-43.208
C02446=1017.024,-25.843,382.374,-24.126,21.559,-43.204
C02447=1017.023,-25.510,382.349,-24.126,21.559,-43.199
C02448=1017.023,-25.177,382.322,-24.127,21.558,-43.195
C02449=1017.021,-24.844,382.295,-24.128,21.558,-43.190
C02450=1017.021,-24.512,382.269,-24.128,21.557,-43.186
C02451=1017.020,-24.179,382.244,-24.129,21.557,-43.181
C02452=1017.019,-23.846,382.217,-24.129,21.556,-43.177
C02453=1017.018,-23.513,382.190,-24.130,21.556,-43.171
C02454=1017.017,-23.180,382.164,-24.131,21.555,-43.168
C02455=1017.016,-22.847,382.138,-24.131,21.556,-43.162
C02456=1017.015,-22.515,382.111,-24.132,21.554,-43.158
C02457=1017.014,-22.182,382.085,-24.133,21.554,-43.153
C02458=1017.013,-21.849,382.058,-24.133,21.554,-43.149
C02459=1017.013,-21.517,382.032,-24.134,21.553,-43.144
C02460=1017.011,-21.183,382.005,-24.134,21.552,-43.140
C02461=1017.011,-20.851,381.979,-24.135,21.553,-43.135
C02462=1017.009,-20.518,381.952,-24.136,21.552,-43.131
C02463=1017.008,-20.185,381.925,-24.136,21.551,-43.127
C02464=1017.008,-19.852,381.899,-24.137,21.551,-43.122
C02465=1017.007,-19.680,381.886,-24.137,21.550,-43.118
C02466=1017.005,-19.263,381.852,-24.138,21.550,-43.112
C02467=1017.005,-19.016,381.832,-24.139,21.550,-43.109
C02468=1017.004,-18.754,381.811,-24.139,21.550,-43.107
C02469=1017.002,-18.492,381.791,-24.139,21.549,-43.105
C02470=1017.002,-18.245,381.771,-24.139,21.548,-43.103
C02471=1017.001,-18.023,381.754,-24.140,21.549,-43.100
C02472=1017.000,-17.658,381.724,-24.141,21.548,-43.092
C02473=1017.000,-17.325,381.697,-24.141,21.547,-43.088
C02474=1016.998,-16.992,381.671,-24.142,21.547,-43.083
C02475=1016.997,-16.659,381.644,-24.142,21.547,-43.079
C02476=1016.995,-16.324,381.617,-24.143,21.546,-43.074
C02477=1016.994,-15.990,381.591,-24.144,21.546,-43.070
C02478=1016.992,-15.656,381.564,-24.145,21.546,-43.065
C02479=1016.992,-15.319,381.536,-24.145,21.545,-43.061
C02480=1016.990,-14.981,381.509,-24.146,21.544,-43.055
C02481=1016.989,-14.641,381.483,-24.146,21.544,-43.052
C02482=1016.987,-14.299,381.454,-24.147,21.544,-43.046
C02483=1016.986,-13.954,381.427,-24.147,21.543,-43.042
C02484=1016.984,-13.608,381.399,-24.148,21.543,-43.037
C02485=1016.983,-13.260,381.372,-24.149,21.542,-43.033
C02486=1016.982,-12.909,381.343,-24.149,21.542,-43.028
C02487=1016.980,-12.558,381.315,-24.150,21.541,-43.024
C02488=1016.978,-12.204,381.286,-24.151,21.541,-43.019
C02489=1016.977,-11.850,381.258,-24.151,21.540,-43.014
C02490=1016.976,-11.493,381.229,-24.152,21.540,-43.009
C02491=1016.974,-11.135,381.200,-24.152,21.539,-43.006
C02492=1016.973,-10.777,381.171,-24.153,21.539,-43.000
C02493=1016.971,-10.416,381.142,-24.154,21.539,-42.995
C02494=1016.969,-10.056,381.113,-24.154,21.538,-42.991
C02495=1016.968,-9.694,381.083,-24.155,21.538,-42.985
C02496=1016.966,-9.332,381.054,-24.156,21.537,-42.982
C02497=1016.965,-8.969,381.025,-24.156,21.536,-42.976
C02498=1016.963,-8.607,380.996,-24.157,21.536,-42.971
C02499=1016.962,-8.244,380.966,-24.158,21.536,-42.967
C02500=1016.959,-7.880,380.937,-24.158,21.535,-42.961
C02501=1016.958,-7.515,380.908,-24.159,21.535,-42.956
C02502=1016.956,-7.145,380.878,-24.160,21.534,-42.952
C02503=1016.954,-6.773,380.847,-24.160,21.534,-42.947
C02504=1016.952,-6.399,380.817,-24.161,21.533,-42.941
C02505=1016.950,-6.023,380.786,-24.162,21.533,-42.937
C02506=1016.948,-5.647,380.756,-24.163,21.533,-42.932
C02507=1016.946,-5.275,380.726,-24.163,21.532,-42.928
C02508=1016.945,-4.904,380.696,-24.164,21.532,-42.923
C02509=1016.942,-4.538,380.666,-24.164,21.531,-42.919
C02510=1016.940,-4.177,380.637,-24.165,21.530,-42.913
C02511=1016.938,-3.819,380.607,-24.166,21.531,-42.908
C02512=1016.937,-3.465,380.579,-24.166,21.529,-42.904
C02513=1016.935,-3.112,380.550,-24.167,21.529,-42.899
C02514=1016.934,-2.893,380.532,-24.167,21.529,-42.897
C02515=1016.932,-2.675,380.514,-24.168,21.529,-42.893
C02516=1016.931,-2.411,380.493,-24.168,21.529,-42.890
C02517=1016.929,-2.063,380.465,-24.169,21.528,-42.886
C02518=1016.927,-1.716,380.436,-24.169,21.528,-42.880
C02519=1016.926,-1.371,380.408,-24.170,21.527,-42.877
C02520=1016.923,-1.028,380.380,-24.170,21.527,-42.873
C02521=1016.921,-0.686,380.352,-24.171,21.526,-42.867
C02522=1016.919,-0.347,380.324,-24.172,21.526,-42.864
C02523=1016.917,-0.007,380.297,-24.172,21.526,-42.858
C02524=1016.915,0.329,380.269,-24.173,21.525,-42.855
C02525=1016.913,0.666,380.242,-24.173,21.525,-42.851
C02526=1016.911,1.000,380.214,-24.174,21.525,-42.846
C02527=1016.909,1.335,380.187,-24.175,21.524,-42.842
C02528=1016.907,1.668,380.159,-24.175,21.523,-42.838
C02529=1016.905,1.998,380.132,-24.176,21.523,-42.834
C02530=1016.904,2.311,380.107,-24.176,21.523,-42.831
C02531=1016.902,2.598,380.083,-24.177,21.522,-42.827
C02532=1016.900,2.868,380.061,-24.177,21.522,-42.823
C02533=1016.899,3.129,380.040,-24.178,21.522,-42.818
C02534=1016.897,3.399,380.017,-24.179,21.521,-42.814
C02535=1016.894,3.688,379.994,-24.179,21.521,-42.810
C02536=1016.893,4.002,379.968,-24.179,21.520,-42.807
C02537=1016.891,4.331,379.941,-24.180,21.521,-42.803
C02538=1016.889,4.663,379.913,-24.180,21.519,-42.799
C02539=1016.886,4.994,379.886,-24.181,21.519,-42.795
C02540=1016.884,5.325,379.859,-24.181,21.518,-42.792
C02541=1016.882,5.655,379.832,-24.182,21.519,-42.786
C02542=1016.880,5.984,379.805,-24.183,21.518,-42.783
C02543=1016.878,6.314,379.777,-24.183,21.518,-42.779
C02544=1016.875,6.643,379.750,-24.184,21.518,-42.774
C02545=1016.873,6.972,379.724,-24.185,21.517,-42.770
C02546=1016.871,7.299,379.696,-24.185,21.517,-42.766
C02547=1016.868,7.625,379.669,-24.186,21.516,-42.762
C02548=1016.867,7.948,379.643,-24.186,21.516,-42.759
C02549=1016.864,8.268,379.616,-24.186,21.515,-42.755
C02550=1016.862,8.586,379.590,-24.187,21.516,-42.750
C02551=1016.860,8.904,379.564,-24.188,21.515,-42.746
C02552=1016.858,9.218,379.538,-24.188,21.515,-42.742
C02553=1016.855,9.533,379.512,-24.189,21.514,-42.738
C02554=1016.854,9.848,379.486,-24.190,21.514,-42.733
C02555=1016.851,10.163,379.460,-24.190,21.514,-42.730
C02556=1016.849,10.480,379.434,-24.191,21.513,-42.726
C02557=1016.846,10.799,379.407,-24.191,21.513,-42.722
C02558=1016.844,11.120,379.381,-24.192,21.512,-42.718
C02559=1016.841,11.442,379.354,-24.192,21.512,-42.715
C02560=1016.840,11.765,379.327,-24.193,21.511,-42.711
C02561=1016.837,12.089,379.301,-24.193,21.511,-42.707
C02562=1016.834,12.412,379.273,-24.194,21.511,-42.702
C02563=1016.832,12.736,379.247,-24.194,21.510,-42.698
C02564=1016.830,13.060,379.220,-24.195,21.510,-42.694
C02565=1016.827,13.383,379.193,-24.195,21.509,-42.691
C02566=1016.825,13.707,379.166,-24.196,21.509,-42.687
C02567=1016.822,14.032,379.139,-24.197,21.509,-42.682
C02568=1016.819,14.356,379.112,-24.197,21.509,-42.678
C02569=1016.817,14.681,379.085,-24.198,21.508,-42.674
C02570=1016.815,15.006,379.058,-24.198,21.508,-42.670
C02571=1016.812,15.333,379.031,-24.199,21.507,-42.667
C02572=1016.810,15.658,379.004,-24.199,21.507,-42.663
C02573=1016.806,15.986,378.977,-24.200,21.507,-42.658
C02574=1016.804,16.314,378.950,-24.200,21.506,-42.654
C02575=1016.801,16.642,378.922,-24.201,21.506,-42.650
C02576=1016.799,16.970,378.894,-24.201,21.505,-42.646
C02577=1016.796,17.300,378.867,-24.202,21.505,-42.643
C02578=1016.793,17.629,378.839,-24.202,21.504,-42.639
C02579=1016.790,17.960,378.812,-24.203,21.504,-42.634
C02580=1016.788,18.291,378.784,-24.204,21.504,-42.630
C02581=1016.785,18.622,378.756,-24.204,21.503,-42.626
C02582=1016.783,18.953,378.729,-24.205,21.503,-42.622
C02583=1016.779,19.286,378.701,-24.205,21.502,-42.619
C02584=1016.776,19.633,378.672,-24.206,21.503,-42.613
C02585=1016.773,20.051,378.637,-24.207,21.502,-42.608
C02586=1016.771,20.287,378.617,-24.207,21.502,-42.604
C02587=1016.769,20.534,378.597,-24.207,21.502,-42.603
C02588=1016.767,20.782,378.576,-24.208,21.502,-42.601
C02589=1016.764,21.024,378.556,-24.208,21.502,-42.599
C02590=1016.763,21.250,378.537,-24.208,21.501,-42.597
C02591=1016.761,21.458,378.520,-24.209,21.501,-42.593
C02592=1016.758,21.815,378.489,-24.209,21.500,-42.588
C02593=1016.754,22.139,378.462,-24.210,21.501,-42.584
C02594=1016.752,22.433,378.438,-24.210,21.500,-42.582
C02595=1016.750,22.686,378.417,-24.210,21.499,-42.580
C02596=1016.746,23.095,378.382,-24.211,21.499,-42.573
C02597=1016.742,23.504,378.348,-24.212,21.498,-42.565
C02598=1016.741,23.756,378.327,-24.213,21.498,-42.562
C02599=1016.738,24.050,378.302,-24.213,21.498,-42.560
C02600=1016.734,24.376,378.275,-24.213,21.497,-42.558
C02601=1016.732,24.710,378.246,-24.214,21.497,-42.553
C02602=1016.728,25.045,378.218,-24.215,21.497,-42.549
C02603=1016.726,25.380,378.191,-24.215,21.496,-42.545
C02604=1016.722,25.713,378.162,-24.216,21.496,-42.541
C02605=1016.719,26.048,378.135,-24.216,21.495,-42.538
C02606=1016.716,26.382,378.106,-24.217,21.495,-42.534
C02607=1016.713,26.716,378.078,-24.217,21.494,-42.530
C02608=1016.710,27.051,378.050,-24.218,21.494,-42.525
C02609=1016.707,27.385,378.021,-24.219,21.495,-42.522
C02610=1016.703,27.719,377.993,-24.219,21.494,-42.518
C02611=1016.700,28.054,377.966,-24.220,21.494,-42.514
C02612=1016.697,28.388,377.937,-24.220,21.493,-42.510
C02613=1016.693,28.722,377.909,-24.221,21.493,-42.507
C02614=1016.690,29.058,377.881,-24.221,21.492,-42.503
C02615=1016.687,29.391,377.853,-24.222,21.493,-42.498
C02616=1016.684,29.726,377.824,-24.222,21.492,-42.494
C02617=1016.680,30.060,377.796,-24.223,21.492,-42.490
C02618=1016.677,30.395,377.767,-24.223,21.491,-42.486
C02619=1016.674,30.729,377.739,-24.224,21.491,-42.483
C02620=1016.670,31.064,377.711,-24.224,21.490,-42.479
C02621=1016.667,31.398,377.682,-24.225,21.490,-42.475
C02622=1016.663,31.733,377.654,-24.225,21.489,-42.471
C02623=1016.660,32.068,377.626,-24.226,21.489,-42.468
C02624=1016.656,32.402,377.598,-24.226,21.489,-42.464
C02625=1016.653,32.737,377.569,-24.227,21.489,-42.459
C02626=1016.650,33.071,377.541,-24.228,21.489,-42.455
C02627=1016.646,33.406,377.513,-24.228,21.488,-42.452
C02628=1016.643,33.740,377.484,-24.229,21.488,-42.448
C02629=1016.639,34.074,377.456,-24.229,21.487,-42.444
C02630=1016.636,34.410,377.428,-24.230,21.487,-42.440
C02631=1016.632,34.744,377.400,-24.230,21.486,-42.437
C02632=1016.629,35.079,377.372,-24.231,21.486,-42.433
C02633=1016.625,35.413,377.342,-24.231,21.485,-42.429
C02634=1016.622,35.748,377.314,-24.232,21.486,-42.426
C02635=1016.618,36.083,377.286,-24.232,21.485,-42.422
C02636=1016.615,36.418,377.258,-24.233,21.485,-42.418
C02637=1016.611,36.752,377.229,-24.234,21.485,-42.413
C02638=1016.607,37.086,377.201,-24.234,21.485,-42.409
C02639=1016.604,37.421,377.172,-24.235,21.484,-42.405
C02640=1016.599,37.756,377.144,-24.235,21.484,-42.402
C02641=1016.596,38.091,377.115,-24.236,21.483,-42.398
C02642=1016.593,38.425,377.087,-24.236,21.483,-42.395
C02643=1016.589,38.760,377.058,-24.237,21.483,-42.391
C02644=1016.585,39.095,377.030,-24.237,21.483,-42.387
C02645=1016.581,39.430,377.001,-24.238,21.482,-42.383
C02646=1016.577,39.765,376.973,-24.238,21.482,-42.380
C02647=1016.574,40.100,376.945,-24.239,21.481,-42.376
C02648=1016.570,40.434,376.916,-24.239,21.481,-42.372
C02649=1016.567,40.769,376.887,-24.240,21.481,-42.369
C02650=1016.562,41.104,376.859,-24.240,21.481,-42.365
C02651=1016.558,41.438,376.830,-24.241,21.480,-42.361
C02652=1016.554,41.774,376.802,-24.241,21.480,-42.357
C02653=1016.550,42.108,376.773,-24.242,21.479,-42.354
C02654=1016.547,42.443,376.745,-24.242,21.479,-42.350
C02655=1016.542,42.777,376.716,-24.243,21.479,-42.347
C02656=1016.539,43.113,376.687,-24.243,21.479,-42.343
C02657=1016.535,43.447,376.659,-24.244,21.478,-42.339
C02658=1016.531,43.783,376.630,-24.244,21.478,-42.335
C02659=1016.526,44.117,376.601,-24.245,21.477,-42.332
C02660=1016.523,44.453,376.573,-24.245,21.477,-42.328
C02661=1016.519,44.787,376.545,-24.246,21.477,-42.325
C02662=1016.514,45.122,376.516,-24.246,21.477,-42.321
C02663=1016.511,45.457,376.486,-24.247,21.476,-42.317
C02664=1016.507,45.791,376.458,-24.247,21.476,-42.313
C02665=1016.503,46.127,376.429,-24.248,21.475,-42.309
C02666=1016.498,46.461,376.401,-24.248,21.475,-42.306
C02667=1016.494,46.796,376.372,-24.249,21.475,-42.302
C02668=1016.490,47.132,376.343,-24.249,21.475,-42.299
C02669=1016.485,47.466,376.315,-24.250,21.474,-42.295
C02670=1016.482,47.801,376.287,-24.250,21.474,-42.291
C02671=1016.478,48.136,376.258,-24.251,21.473,-42.287
C02672=1016.474,48.472,376.229,-24.251,21.473,-42.284
C02673=1016.470,48.806,376.200,-24.252,21.473,-42.280
C02674=1016.465,49.140,376.171,-24.252,21.473,-42.277
C02675=1016.461,49.476,376.142,-24.253,21.472,-42.273
C02676=1016.457,49.811,376.114,-24.253,21.472,-42.269
C02677=1016.452,50.145,376.085,-24.254,21.472,-42.266
C02678=1016.448,50.481,376.056,-24.254,21.471,-42.262
C02679=1016.444,50.815,376.028,-24.255,21.471,-42.258
C02680=1016.440,51.151,375.999,-24.255,21.471,-42.254
C02681=1016.435,51.486,375.970,-24.256,21.471,-42.251
C02682=1016.430,51.821,375.941,-24.256,21.470,-42.247
C02683=1016.426,52.156,375.912,-24.257,21.470,-42.244
C02684=1016.422,52.491,375.884,-24.257,21.470,-42.240
C02685=1016.417,52.825,375.855,-24.258,21.469,-42.238
C02686=1016.413,53.161,375.826,-24.258,21.469,-42.234
C02687=1016.409,53.496,375.798,-24.259,21.468,-42.230
C02688=1016.404,53.830,375.768,-24.259,21.468,-42.227
C02689=1016.399,54.165,375.739,-24.260,21.468,-42.223
C02690=1016.395,54.500,375.711,-24.260,21.468,-42.220
C02691=1016.391,54.835,375.682,-24.261,21.467,-42.216
C02692=1016.386,55.170,375.653,-24.261,21.467,-42.212
C02693=1016.382,55.505,375.624,-24.262,21.467,-42.209
C02694=1016.377,55.840,375.595,-24.262,21.467,-42.205
C02695=1016.372,56.175,375.566,-24.263,21.466,-42.201
C02696=1016.367,56.510,375.538,-24.263,21.466,-42.197
C02697=1016.363,56.845,375.509,-24.264,21.466,-42.194
C02698=1016.358,57.180,375.480,-24.264,21.465,-42.192
C02699=1016.354,57.515,375.451,-24.264,21.465,-42.188
C02700=1016.349,57.850,375.423,-24.265,21.464,-42.184
C02701=1016.344,58.185,375.393,-24.266,21.465,-42.181
C02702=1016.340,58.520,375.365,-24.266,21.464,-42.177
C02703=1016.335,58.855,375.335,-24.267,21.464,-42.173
C02704=1016.330,59.190,375.307,-24.267,21.464,-42.170
C02705=1016.325,59.525,375.278,-24.268,21.464,-42.166
C02706=1016.320,59.860,375.249,-24.268,21.463,-42.163
C02707=1016.316,60.195,375.220,-24.268,21.462,-42.160
C02708=1016.311,60.530,375.191,-24.269,21.462,-42.157
C02709=1016.306,60.865,375.162,-24.269,21.462,-42.153
C02710=1016.302,61.199,375.133,-24.270,21.461,-42.149
C02711=1016.297,61.534,375.104,-24.270,21.462,-42.146
C02712=1016.291,61.869,375.075,-24.271,21.461,-42.142
C02713=1016.287,62.204,375.046,-24.271,21.461,-42.139
C02714=1016.282,62.540,375.017,-24.272,21.460,-42.135
C02715=1016.276,62.937,374.983,-24.272,21.460,-42.131
C02716=1016.273,63.161,374.963,-24.273,21.461,-42.130
C02717=1016.270,63.379,374.945,-24.273,21.460,-42.128
C02718=1016.267,63.753,374.911,-24.274,21.460,-42.124
C02719=1016.266,64.109,374.877,-24.274,21.459,-42.120
C02720=1016.264,64.494,374.840,-24.274,21.459,-42.116
C02721=1016.263,64.890,374.803,-24.275,21.458,-42.113
C02722=1016.262,65.267,374.768,-24.276,21.459,-42.108
C02723=1016.261,65.621,374.734,-24.276,21.457,-42.105
C02724=1016.260,65.960,374.703,-24.277,21.458,-42.102
C02725=1016.260,66.294,374.672,-24.277,21.457,-42.098
C02726=1016.258,66.629,374.640,-24.278,21.457,-42.094
C02727=1016.257,66.966,374.608,-24.278,21.457,-42.091
C02728=1016.256,67.303,374.576,-24.279,21.457,-42.087
C02729=1016.255,67.642,374.544,-24.279,21.456,-42.085
C02730=1016.254,67.981,374.512,-24.279,21.456,-42.082
C02731=1016.253,68.321,374.480,-24.280,21.456,-42.078
C02732=1016.252,68.662,374.448,-24.280,21.455,-42.074
C02733=1016.251,69.005,374.415,-24.281,21.456,-42.071
C02734=1016.250,69.347,374.383,-24.281,21.455,-42.067
C02735=1016.249,69.692,374.350,-24.282,21.455,-42.063
C02736=1016.248,70.036,374.317,-24.282,21.454,-42.061
C02737=1016.247,70.381,374.285,-24.283,21.454,-42.058
C02738=1016.245,70.725,374.253,-24.283,21.453,-42.054
C02739=1016.245,71.070,374.220,-24.284,21.454,-42.051
C02740=1016.243,71.414,374.187,-24.284,21.453,-42.047
C02741=1016.243,71.759,374.154,-24.285,21.453,-42.043
C02742=1016.241,72.104,374.122,-24.285,21.453,-42.041
C02743=1016.240,72.451,374.089,-24.285,21.452,-42.037
C02744=1016.239,72.798,374.056,-24.286,21.452,-42.034
C02745=1016.239,73.148,374.023,-24.286,21.451,-42.030
C02746=1016.237,73.499,373.989,-24.287,21.452,-42.027
C02747=1016.236,73.853,373.956,-24.288,21.451,-42.023
C02748=1016.235,74.208,373.922,-24.288,21.451,-42.019
C02749=1016.234,74.565,373.888,-24.288,21.451,-42.017
C02750=1016.233,74.923,373.853,-24.289,21.450,-42.013
C02751=1016.232,75.281,373.820,-24.289,21.450,-42.010
C02752=1016.230,75.634,373.786,-24.290,21.450,-42.006
C02753=1016.229,75.983,373.752,-24.290,21.449,-42.004
C02754=1016.228,76.325,373.720,-24.291,21.449,-42.001
C02755=1016.227,76.661,373.687,-24.291,21.449,-41.997
C02756=1016.226,76.991,373.656,-24.292,21.449,-41.994
C02757=1016.225,77.318,373.625,-24.292,21.449,-41.990
C02758=1016.224,77.641,373.594,-24.292,21.448,-41.987
C02759=1016.223,77.965,373.563,-24.293,21.448,-41.984
C02760=1016.221,78.290,373.532,-24.293,21.448,-41.980
C02761=1016.220,78.617,373.500,-24.294,21.447,-41.977
C02762=1016.220,78.950,373.469,-24.295,21.448,-41.973
C02763=1016.218,79.289,373.436,-24.295,21.446,-41.971
C02764=1016.217,79.634,373.403,-24.295,21.447,-41.968
C02765=1016.216,79.985,373.369,-24.296,21.446,-41.964
C02766=1016.215,80.340,373.335,-24.296,21.446,-41.962
C02767=1016.213,80.697,373.301,-24.297,21.446,-41.958
C02768=1016.212,81.054,373.267,-24.297,21.445,-41.955
C02769=1016.212,81.409,373.233,-24.298,21.446,-41.951
C02770=1016.209,81.764,373.199,-24.298,21.445,-41.947
C02771=1016.209,82.119,373.164,-24.298,21.444,-41.945
C02772=1016.207,82.473,373.130,-24.299,21.444,-41.942
C02773=1016.206,82.826,373.097,-24.299,21.444,-41.938
C02774=1016.205,83.177,373.063,-24.300,21.444,-41.935
C02775=1016.204,83.529,373.029,-24.300,21.444,-41.931
C02776=1016.203,83.878,372.996,-24.301,21.443,-41.929
C02777=1016.202,84.227,372.962,-24.301,21.443,-41.925
C02778=1016.201,84.576,372.928,-24.302,21.443,-41.922
C02779=1016.200,84.922,372.895,-24.302,21.443,-41.918
C02780=1016.198,85.267,372.861,-24.302,21.442,-41.916
C02781=1016.197,85.612,372.828,-24.303,21.442,-41.912
C02782=1016.196,85.954,372.795,-24.303,21.442,-41.909
C02783=1016.194,86.297,372.762,-24.304,21.441,-41.906
C02784=1016.193,86.637,372.728,-24.304,21.441,-41.903
C02785=1016.193,86.976,372.696,-24.305,21.441,-41.899
C02786=1016.191,87.314,372.664,-24.305,21.441,-41.898
C02787=1016.190,87.646,372.631,-24.305,21.440,-41.894
C02788=1016.189,87.972,372.599,-24.306,21.441,-41.890
C02789=1016.188,88.294,372.568,-24.306,21.439,-41.888
C02790=1016.187,88.615,372.538,-24.307,21.440,-41.885
C02791=1016.185,88.936,372.506,-24.307,21.439,-41.881
C02792=1016.184,89.261,372.475,-24.308,21.439,-41.879
C02793=1016.183,89.590,372.443,-24.308,21.440,-41.876
C02794=1016.182,89.923,372.410,-24.308,21.438,-41.874
C02795=1016.181,90.258,372.378,-24.309,21.439,-41.870
C02796=1016.179,90.592,372.345,-24.309,21.438,-41.866
C02797=1016.178,90.926,372.313,-24.310,21.438,-41.865
C02798=1016.177,91.261,372.280,-24.310,21.438,-41.861
C02799=1016.176,91.595,372.248,-24.311,21.438,-41.857
C02800=1016.175,91.930,372.216,-24.311,21.437,-41.855
C02801=1016.173,92.264,372.183,-24.311,21.437,-41.852
C02802=1016.172,92.598,372.151,-24.312,21.436,-41.849
C02803=1016.171,92.934,372.118,-24.312,21.437,-41.846
C02804=1016.169,93.268,372.085,-24.313,21.436,-41.842
C02805=1016.169,93.601,372.053,-24.313,21.436,-41.841
C02806=1016.168,93.936,372.020,-24.314,21.436,-41.837
C02807=1016.166,94.270,371.988,-24.314,21.436,-41.833
C02808=1016.165,94.605,371.955,-24.314,21.436,-41.832
C02809=1016.164,94.939,371.922,-24.315,21.435,-41.828
C02810=1016.162,95.274,371.890,-24.315,21.435,-41.826
C02811=1016.161,95.607,371.857,-24.316,21.435,-41.822
C02812=1016.160,95.941,371.825,-24.316,21.435,-41.819
C02813=1016.159,96.276,371.792,-24.316,21.434,-41.817
C02814=1016.157,96.610,371.760,-24.317,21.434,-41.813
C02815=1016.157,96.945,371.726,-24.317,21.434,-41.811
C02816=1016.155,97.279,371.694,-24.318,21.434,-41.808
C02817=1016.154,97.613,371.661,-24.318,21.433,-41.806
C02818=1016.153,97.947,371.628,-24.318,21.433,-41.802
C02819=1016.151,98.281,371.595,-24.319,21.433,-41.799
C02820=1016.150,98.616,371.563,-24.319,21.432,-41.796
C02821=1016.148,98.949,371.530,-24.320,21.433,-41.793
C02822=1016.148,99.283,371.498,-24.320,21.432,-41.791
C02823=1016.146,99.618,371.465,-24.320,21.432,-41.787
C02824=1016.146,99.952,371.432,-24.321,21.432,-41.785
C02825=1016.144,100.287,371.399,-24.321,21.431,-41.782
C02826=1016.143,100.620,371.366,-24.322,21.432,-41.778
C02827=1016.141,100.955,371.333,-24.322,21.431,-41.776
C02828=1016.140,101.288,371.300,-24.323,21.431,-41.773
C02829=1016.139,101.623,371.268,-24.323,21.431,-41.771
C02830=1016.137,101.957,371.235,-24.323,21.430,-41.767
C02831=1016.136,102.291,371.202,-24.324,21.430,-41.765
C02832=1016.135,102.625,371.169,-24.324,21.431,-41.762
C02833=1016.133,102.959,371.136,-24.324,21.429,-41.760
C02834=1016.133,103.294,371.103,-24.325,21.430,-41.756
C02835=1016.131,103.628,371.070,-24.325,21.429,-41.752
C02836=1016.130,103.961,371.037,-24.326,21.429,-41.751
C02837=1016.129,104.296,371.004,-24.326,21.430,-41.747
C02838=1016.128,104.629,370.971,-24.326,21.428,-41.745
C02839=1016.126,104.964,370.939,-24.327,21.429,-41.742
C02840=1016.125,105.297,370.905,-24.327,21.428,-41.739
C02841=1016.123,105.632,370.873,-24.328,21.428,-41.736
C02842=1016.122,105.965,370.840,-24.328,21.428,-41.734
C02843=1016.121,106.299,370.806,-24.328,21.427,-41.730
C02844=1016.120,106.634,370.774,-24.329,21.427,-41.728
C02845=1016.118,106.967,370.741,-24.329,21.428,-41.725
C02846=1016.117,107.302,370.707,-24.329,21.427,-41.723
C02847=1016.116,107.636,370.674,-24.330,21.427,-41.719
C02848=1016.114,107.970,370.641,-24.330,21.427,-41.718
C02849=1016.113,108.304,370.608,-24.331,21.426,-41.714
C02850=1016.112,108.638,370.575,-24.331,21.426,-41.712
C02851=1016.111,108.972,370.542,-24.332,21.426,-41.708
C02852=1016.109,109.306,370.509,-24.332,21.425,-41.706
C02853=1016.108,109.640,370.476,-24.332,21.426,-41.703
C02854=1016.107,109.974,370.443,-24.333,21.425,-41.701
C02855=1016.105,110.308,370.409,-24.333,21.425,-41.697
C02856=1016.104,110.641,370.376,-24.333,21.425,-41.695
C02857=1016.102,110.975,370.343,-24.334,21.424,-41.692
C02858=1016.101,111.309,370.310,-24.334,21.424,-41.690
C02859=1016.100,111.644,370.277,-24.335,21.425,-41.686
C02860=1016.099,111.978,370.243,-24.335,21.423,-41.684
C02861=1016.097,112.312,370.210,-24.335,21.424,-41.681
C02862=1016.096,112.646,370.177,-24.336,21.424,-41.679
C02863=1016.095,112.980,370.144,-24.336,21.423,-41.675
C02864=1016.093,113.313,370.111,-24.336,21.423,-41.673
C02865=1016.092,113.647,370.077,-24.337,21.423,-41.670
C02866=1016.091,113.981,370.044,-24.337,21.422,-41.668
C02867=1016.089,114.315,370.010,-24.338,21.423,-41.664
C02868=1016.088,114.649,369.977,-24.338,21.422,-41.662
C02869=1016.087,114.983,369.945,-24.338,21.421,-41.660
C02870=1016.086,115.317,369.911,-24.339,21.422,-41.657
C02871=1016.084,115.651,369.877,-24.339,21.422,-41.655
C02872=1016.083,115.985,369.844,-24.340,21.422,-41.652
C02873=1016.082,116.319,369.811,-24.340,21.421,-41.649
C02874=1016.080,116.653,369.778,-24.340,21.421,-41.646
C02875=1016.079,116.987,369.744,-24.341,21.421,-41.644
C02876=1016.077,117.320,369.711,-24.341,21.421,-41.640
C02877=1016.076,117.654,369.677,-24.341,21.420,-41.638
C02878=1016.075,117.989,369.643,-24.342,21.421,-41.635
C02879=1016.074,118.323,369.610,-24.342,21.420,-41.633
C02880=1016.073,118.656,369.577,-24.342,21.419,-41.631
C02881=1016.071,118.990,369.543,-24.343,21.420,-41.628
C02882=1016.069,119.324,369.510,-24.343,21.419,-41.625
C02883=1016.068,119.658,369.476,-24.344,21.419,-41.622
C02884=1016.066,119.992,369.443,-24.344,21.419,-41.620
C02885=1016.066,120.326,369.409,-24.345,21.419,-41.617
C02886=1016.065,120.660,369.376,-24.345,21.418,-41.614
C02887=1016.063,120.994,369.342,-24.345,21.418,-41.613
C02888=1016.061,121.328,369.309,-24.346,21.418,-41.609
C02889=1016.060,121.662,369.275,-24.346,21.417,-41.607
C02890=1016.058,121.995,369.242,-24.346,21.418,-41.604
C02891=1016.058,122.330,369.208,-24.347,21.418,-41.602
C02892=1016.056,122.664,369.174,-24.347,21.418,-41.598
C02893=1016.055,122.998,369.141,-24.347,21.417,-41.596
C02894=1016.053,123.332,369.107,-24.348,21.417,-41.594
C02895=1016.052,123.666,369.074,-24.348,21.417,-41.591
C02896=1016.050,124.000,369.040,-24.348,21.417,-41.589
C02897=1016.049,124.334,369.007,-24.349,21.416,-41.585
C02898=1016.048,124.668,368.974,-24.349,21.416,-41.583
C02899=1016.046,125.001,368.939,-24.349,21.416,-41.581
C02900=1016.046,125.335,368.905,-24.350,21.416,-41.578
C02901=1016.044,125.669,368.872,-24.350,21.415,-41.576
C02902=1016.043,126.003,368.838,-24.351,21.416,-41.572
C02903=1016.041,126.337,368.805,-24.351,21.415,-41.571
C02904=1016.040,126.672,368.771,-24.351,21.415,-41.569
C02905=1016.038,127.006,368.737,-24.352,21.415,-41.565
C02906=1016.036,127.340,368.703,-24.352,21.415,-41.563
C02907=1016.036,127.673,368.669,-24.352,21.414,-41.561
C02908=1016.034,128.007,368.635,-24.353,21.415,-41.558
C02909=1016.033,128.341,368.602,-24.353,21.414,-41.555
C02910=1016.032,128.676,368.568,-24.354,21.414,-41.552
C02911=1016.030,129.010,368.535,-24.354,21.414,-41.550
C02912=1016.029,129.344,368.501,-24.354,21.414,-41.548
C02913=1016.028,129.678,368.466,-24.355,21.413,-41.545
C02914=1016.026,130.012,368.433,-24.355,21.413,-41.543
C02915=1016.024,130.346,368.399,-24.355,21.413,-41.541
C02916=1016.024,130.680,368.365,-24.356,21.413,-41.538
C02917=1016.022,131.014,368.331,-24.356,21.412,-41.535
C02918=1016.021,131.348,368.297,-24.356,21.412,-41.532
C02919=1016.020,131.682,368.263,-24.357,21.412,-41.530
C02920=1016.018,132.016,368.230,-24.357,21.412,-41.528
C02921=1016.017,132.351,368.195,-24.357,21.412,-41.525
C02922=1016.015,132.684,368.162,-24.358,21.411,-41.523
C02923=1016.014,133.019,368.127,-24.358,21.411,-41.521
C02924=1016.012,133.353,368.093,-24.358,21.411,-41.517
C02925=1016.011,133.687,368.059,-24.359,21.411,-41.515
C02926=1016.010,134.021,368.026,-24.359,21.410,-41.513
C02927=1016.008,134.354,367.991,-24.359,21.411,-41.510
C02928=1016.007,134.689,367.957,-24.360,21.410,-41.508
C02929=1016.005,135.023,367.923,-24.360,21.410,-41.506
C02930=1016.004,135.356,367.890,-24.361,21.411,-41.503
C02931=1016.003,135.679,367.857,-24.361,21.410,-41.501
C02932=1016.001,135.981,367.826,-24.361,21.410,-41.499
C02933=1016.001,136.259,367.798,-24.361,21.410,-41.497
C02934=1016.000,136.524,367.770,-24.361,21.409,-41.495
C02935=1015.999,136.789,367.744,-24.362,21.409,-41.491
C02936=1015.998,137.065,367.715,-24.362,21.409,-41.490
C02937=1015.996,137.362,367.685,-24.363,21.409,-41.488
C02938=1015.995,137.684,367.653,-24.363,21.408,-41.486
C02939=1015.993,138.024,367.618,-24.363,21.408,-41.484
C02940=1015.992,138.381,367.581,-24.364,21.408,-41.480
C02941=1015.990,138.792,367.538,-24.364,21.408,-41.477
C02942=1015.990,139.020,367.516,-24.364,21.408,-41.475
C02943=1015.988,139.257,367.492,-24.365,21.408,-41.473
C02944=1015.987,139.500,367.467,-24.365,21.408,-41.473
C02945=1015.986,139.740,367.442,-24.365,21.408,-41.471
C02946=1015.986,139.973,367.418,-24.365,21.408,-41.470
C02947=1015.985,140.194,367.395,-24.365,21.407,-41.469
C02948=1015.983,140.587,367.355,-24.366,21.407,-41.465
C02949=1015.982,140.932,367.320,-24.366,21.407,-41.462
C02950=1015.980,141.271,367.285,-24.367,21.407,-41.460
C02951=1015.979,141.611,367.250,-24.367,21.407,-41.457
C02952=1015.978,141.951,367.215,-24.367,21.406,-41.455
C02953=1015.976,142.291,367.181,-24.368,21.406,-41.453
C02954=1015.975,142.632,367.145,-24.368,21.407,-41.449
C02955=1015.974,142.975,367.110,-24.368,21.406,-41.448
C02956=1015.972,143.318,367.075,-24.369,21.405,-41.445
C02957=1015.971,143.660,367.040,-24.369,21.406,-41.442
C02958=1015.969,144.004,367.004,-24.369,21.405,-41.440
C02959=1015.968,144.349,366.969,-24.370,21.405,-41.438
C02960=1015.967,144.692,366.934,-24.370,21.406,-41.435
C02961=1015.965,145.038,366.899,-24.370,21.405,-41.432
C02962=1015.964,145.383,366.862,-24.371,21.404,-41.431
C02963=1015.962,145.728,366.827,-24.371,21.405,-41.427
C02964=1015.962,146.075,366.791,-24.371,21.405,-41.425
C02965=1015.960,146.420,366.756,-24.372,21.404,-41.424
C02966=1015.958,146.768,366.720,-24.372,21.404,-41.420
C02967=1015.946,147.113,366.691,-24.372,21.404,-41.418
C02968=1016.346,147.142,366.441,-24.372,21.404,-41.418
C02969=1016.360,146.796,366.469,-24.372,21.404,-41.420
C02970=1016.362,146.450,366.505,-24.372,21.404,-41.424
C02971=1016.364,146.104,366.540,-24.371,21.405,-41.425
C02972=1016.365,145.758,366.576,-24.371,21.405,-41.427
C02973=1016.366,145.412,366.611,-24.371,21.404,-41.431
C02974=1016.367,145.067,366.647,-24.370,21.405,-41.432
C02975=1016.369,144.722,366.683,-24.370,21.406,-41.435
C02976=1016.370,144.378,366.718,-24.370,21.405,-41.438
C02977=1016.371,144.033,366.754,-24.369,21.405,-41.440
C02978=1016.373,143.690,366.789,-24.369,21.406,-41.442
C02979=1016.374,143.346,366.825,-24.369,21.405,-41.445
C02980=1016.375,143.004,366.860,-24.368,21.406,-41.448
C02981=1016.377,142.662,366.895,-24.368,21.407,-41.449
C02982=1016.379,142.320,366.930,-24.368,21.406,-41.453
C02983=1016.379,141.980,366.965,-24.367,21.406,-41.455
C02984=1016.381,141.639,366.999,-24.367,21.407,-41.457
C02985=1016.383,141.300,367.034,-24.367,21.407,-41.460
C02986=1016.384,140.961,367.069,-24.366,21.407,-41.462
C02987=1016.385,140.616,367.105,-24.366,21.407,-41.465
C02988=1016.387,140.223,367.145,-24.365,21.407,-41.469
C02989=1016.387,140.002,367.168,-24.365,21.408,-41.470
C02990=1016.388,139.769,367.191,-24.365,21.408,-41.471
C02991=1016.389,139.529,367.216,-24.365,21.408,-41.473
C02992=1016.390,139.287,367.240,-24.365,21.408,-41.473
C02993=1016.391,139.049,367.265,-24.364,21.408,-41.475
C02994=1016.392,138.821,367.288,-24.364,21.408,-41.477
C02995=1016.394,138.410,367.330,-24.364,21.408,-41.480
C02996=1016.396,138.053,367.367,-24.363,21.408,-41.484
C02997=1016.397,137.713,367.402,-24.363,21.408,-41.486
C02998=1016.398,137.391,367.434,-24.363,21.409,-41.488
C02999=1016.399,137.094,367.465,-24.362,21.409,-41.490
C03000=1016.400,136.818,367.492,-24.362,21.409,-41.491
C03001=1016.402,136.554,367.520,-24.361,21.409,-41.495
C03002=1016.402,136.288,367.547,-24.361,21.410,-41.497
C03003=1016.403,136.009,367.575,-24.361,21.410,-41.499
C03004=1016.405,135.709,367.606,-24.361,21.410,-41.501
C03005=1016.406,135.386,367.639,-24.361,21.411,-41.503
C03006=1016.408,135.052,367.673,-24.360,21.410,-41.506
C03007=1016.409,134.718,367.707,-24.360,21.410,-41.508
C03008=1016.411,134.384,367.741,-24.359,21.411,-41.510
C03009=1016.411,134.050,367.775,-24.359,21.410,-41.513
C03010=1016.413,133.716,367.809,-24.359,21.411,-41.515
C03011=1016.414,133.382,367.844,-24.358,21.411,-41.517
C03012=1016.416,133.048,367.877,-24.358,21.411,-41.521
C03013=1016.417,132.713,367.911,-24.358,21.411,-41.523
C03014=1016.418,132.379,367.945,-24.357,21.412,-41.525
C03015=1016.419,132.045,367.980,-24.357,21.412,-41.528
C03016=1016.421,131.711,368.013,-24.357,21.412,-41.530
C03017=1016.423,131.377,368.047,-24.356,21.412,-41.532
C03018=1016.424,131.043,368.081,-24.356,21.412,-41.535
C03019=1016.425,130.709,368.114,-24.356,21.413,-41.538
C03020=1016.426,130.375,368.149,-24.355,21.413,-41.541
C03021=1016.427,130.041,368.182,-24.355,21.413,-41.543
C03022=1016.429,129.707,368.216,-24.355,21.413,-41.545
C03023=1016.430,129.372,368.250,-24.354,21.414,-41.548
C03024=1016.431,129.039,368.284,-24.354,21.414,-41.550
C03025=1016.433,128.704,368.318,-24.354,21.414,-41.552
C03026=1016.434,128.371,368.352,-24.353,21.414,-41.555
C03027=1016.436,128.037,368.385,-24.353,21.415,-41.558
C03028=1016.438,127.703,368.419,-24.352,21.414,-41.561
C03029=1016.438,127.368,368.453,-24.352,21.415,-41.563
C03030=1016.440,127.035,368.487,-24.352,21.415,-41.565
C03031=1016.441,126.701,368.520,-24.351,21.415,-41.569
C03032=1016.442,126.366,368.555,-24.351,21.415,-41.571
C03033=1016.444,126.033,368.588,-24.351,21.416,-41.572
C03034=1016.445,125.699,368.622,-24.350,21.415,-41.576
C03035=1016.446,125.364,368.655,-24.350,21.416,-41.578
C03036=1016.448,125.030,368.689,-24.349,21.416,-41.581
C03037=1016.449,124.696,368.722,-24.349,21.416,-41.583
C03038=1016.451,124.363,368.757,-24.349,21.416,-41.585
C03039=1016.451,124.029,368.790,-24.348,21.417,-41.589
C03040=1016.452,123.695,368.824,-24.348,21.417,-41.591
C03041=1016.454,123.361,368.857,-24.348,21.417,-41.594
C03042=1016.456,123.027,368.891,-24.347,21.417,-41.596
C03043=1016.457,122.692,368.925,-24.347,21.418,-41.598
C03044=1016.458,122.359,368.958,-24.347,21.418,-41.602
C03045=1016.460,122.025,368.992,-24.346,21.418,-41.604
C03046=1016.461,121.691,369.025,-24.346,21.417,-41.607
C03047=1016.462,121.357,369.058,-24.346,21.418,-41.609
C03048=1016.464,121.022,369.093,-24.345,21.418,-41.613
C03049=1016.465,120.689,369.126,-24.345,21.418,-41.614
C03050=1016.466,120.355,369.159,-24.345,21.419,-41.617
C03051=1016.468,120.021,369.193,-24.344,21.419,-41.620
C03052=1016.469,119.687,369.226,-24.344,21.419,-41.622
C03053=1016.470,119.353,369.259,-24.343,21.419,-41.625
C03054=1016.472,119.019,369.293,-24.343,21.420,-41.628
C03055=1016.473,118.685,369.327,-24.342,21.419,-41.631
C03056=1016.474,118.351,369.360,-24.342,21.420,-41.633
C03057=1016.476,118.017,369.394,-24.342,21.421,-41.635
C03058=1016.477,117.684,369.427,-24.341,21.420,-41.638
C03059=1016.478,117.350,369.460,-24.341,21.421,-41.640
C03060=1016.480,117.016,369.494,-24.341,21.421,-41.644
C03061=1016.481,116.681,369.527,-24.340,21.421,-41.646
C03062=1016.482,116.348,369.561,-24.340,21.421,-41.649
C03063=1016.483,116.014,369.594,-24.340,21.422,-41.652
C03064=1016.485,115.680,369.628,-24.339,21.422,-41.655
C03065=1016.486,115.346,369.661,-24.339,21.422,-41.657
C03066=1016.487,115.012,369.694,-24.338,21.421,-41.660
C03067=1016.489,114.679,369.727,-24.338,21.422,-41.662
C03068=1016.490,114.344,369.762,-24.338,21.423,-41.664
C03069=1016.491,114.010,369.794,-24.337,21.422,-41.668
C03070=1016.493,113.676,369.827,-24.337,21.423,-41.670
C03071=1016.494,113.342,369.861,-24.336,21.423,-41.673
C03072=1016.495,113.008,369.894,-24.336,21.423,-41.675
C03073=1016.497,112.674,369.928,-24.336,21.424,-41.679
C03074=1016.498,112.341,369.961,-24.335,21.424,-41.681
C03075=1016.499,112.006,369.993,-24.335,21.423,-41.684
C03076=1016.501,111.673,370.027,-24.335,21.425,-41.686
C03077=1016.502,111.339,370.060,-24.334,21.424,-41.690
C03078=1016.503,111.004,370.094,-24.334,21.424,-41.692
C03079=1016.504,110.670,370.127,-24.333,21.425,-41.695
C03080=1016.506,110.336,370.160,-24.333,21.425,-41.697
C03081=1016.507,110.002,370.193,-24.333,21.425,-41.701
C03082=1016.508,109.669,370.226,-24.332,21.426,-41.703
C03083=1016.509,109.335,370.259,-24.332,21.425,-41.706
C03084=1016.511,109.001,370.292,-24.332,21.426,-41.708
C03085=1016.512,108.667,370.325,-24.331,21.426,-41.712
C03086=1016.513,108.333,370.358,-24.331,21.426,-41.714
C03087=1016.515,107.999,370.392,-24.330,21.427,-41.718
C03088=1016.517,107.665,370.425,-24.330,21.427,-41.719
C03089=1016.517,107.330,370.458,-24.329,21.427,-41.723
C03090=1016.518,106.997,370.491,-24.329,21.428,-41.725
C03091=1016.520,106.662,370.524,-24.329,21.427,-41.728
C03092=1016.521,106.329,370.557,-24.328,21.427,-41.730
C03093=1016.522,105.995,370.590,-24.328,21.428,-41.734
C03094=1016.524,105.661,370.623,-24.328,21.428,-41.736
C03095=1016.525,105.327,370.656,-24.327,21.428,-41.739
C03096=1016.526,104.992,370.689,-24.327,21.429,-41.742
C03097=1016.528,104.659,370.722,-24.326,21.428,-41.745
C03098=1016.529,104.325,370.755,-24.326,21.430,-41.747
C03099=1016.530,103.991,370.787,-24.326,21.429,-41.751
C03100=1016.531,103.656,370.821,-24.325,21.429,-41.752
C03101=1016.532,103.322,370.854,-24.325,21.430,-41.756
C03102=1016.533,102.988,370.887,-24.324,21.429,-41.760
C03103=1016.535,102.654,370.919,-24.324,21.431,-41.762
C03104=1016.536,102.320,370.953,-24.324,21.430,-41.765
C03105=1016.538,101.986,370.985,-24.323,21.430,-41.767
C03106=1016.539,101.652,371.018,-24.323,21.431,-41.771
C03107=1016.540,101.318,371.051,-24.323,21.431,-41.773
C03108=1016.541,100.984,371.084,-24.322,21.431,-41.776
C03109=1016.543,100.650,371.116,-24.322,21.432,-41.778
C03110=1016.543,100.315,371.150,-24.321,21.431,-41.782
C03111=1016.545,99.981,371.183,-24.321,21.432,-41.785
C03112=1016.546,99.647,371.215,-24.320,21.432,-41.787
C03113=1016.548,99.313,371.248,-24.320,21.432,-41.791
C03114=1016.549,98.978,371.281,-24.320,21.433,-41.793
C03115=1016.550,98.645,371.314,-24.319,21.432,-41.796
C03116=1016.551,98.311,371.346,-24.319,21.433,-41.799
C03117=1016.553,97.976,371.378,-24.318,21.433,-41.802
C03118=1016.553,97.642,371.412,-24.318,21.433,-41.806
C03119=1016.555,97.308,371.444,-24.318,21.434,-41.808
C03120=1016.556,96.973,371.477,-24.317,21.434,-41.811
C03121=1016.557,96.640,371.510,-24.317,21.434,-41.813
C03122=1016.559,96.305,371.543,-24.316,21.434,-41.817
C03123=1016.560,95.971,371.575,-24.316,21.435,-41.819
C03124=1016.561,95.636,371.608,-24.316,21.435,-41.822
C03125=1016.562,95.302,371.640,-24.315,21.435,-41.826
C03126=1016.563,94.968,371.673,-24.315,21.435,-41.828
C03127=1016.565,94.634,371.706,-24.314,21.436,-41.832
C03128=1016.566,94.299,371.738,-24.314,21.436,-41.833
C03129=1016.567,93.965,371.771,-24.314,21.436,-41.837
C03130=1016.568,93.630,371.804,-24.313,21.436,-41.841
C03131=1016.570,93.296,371.837,-24.313,21.436,-41.842
C03132=1016.570,92.962,371.869,-24.312,21.437,-41.846
C03133=1016.572,92.628,371.901,-24.312,21.436,-41.849
C03134=1016.573,92.293,371.934,-24.311,21.437,-41.852
C03135=1016.574,91.958,371.967,-24.311,21.437,-41.855
C03136=1016.576,91.624,371.999,-24.311,21.438,-41.857
C03137=1016.576,91.290,372.031,-24.310,21.438,-41.861
C03138=1016.578,90.956,372.064,-24.310,21.438,-41.865
C03139=1016.579,90.621,372.096,-24.309,21.438,-41.866
C03140=1016.580,90.286,372.129,-24.309,21.439,-41.870
C03141=1016.582,89.952,372.161,-24.308,21.438,-41.874
C03142=1016.583,89.619,372.194,-24.308,21.440,-41.876
C03143=1016.584,89.290,372.226,-24.308,21.439,-41.879
C03144=1016.585,88.965,372.257,-24.307,21.439,-41.881
C03145=1016.586,88.644,372.289,-24.307,21.440,-41.885
C03146=1016.587,88.324,372.320,-24.306,21.439,-41.888
C03147=1016.588,88.001,372.350,-24.306,21.441,-41.890
C03148=1016.589,87.675,372.382,-24.305,21.440,-41.894
C03149=1016.590,87.342,372.415,-24.305,21.441,-41.898
C03150=1016.591,87.005,372.446,-24.305,21.441,-41.899
C03151=1016.593,86.666,372.480,-24.304,21.441,-41.903
C03152=1016.594,86.325,372.513,-24.304,21.441,-41.906
C03153=1016.595,85.983,372.546,-24.303,21.442,-41.909
C03154=1016.596,85.641,372.579,-24.303,21.442,-41.912
C03155=1016.597,85.296,372.612,-24.302,21.442,-41.916
C03156=1016.599,84.951,372.646,-24.302,21.443,-41.918
C03157=1016.600,84.604,372.679,-24.302,21.443,-41.922
C03158=1016.600,84.256,372.712,-24.301,21.443,-41.925
C03159=1016.602,83.907,372.746,-24.301,21.443,-41.929
C03160=1016.604,83.557,372.780,-24.300,21.444,-41.931
C03161=1016.605,83.206,372.814,-24.300,21.444,-41.935
C03162=1016.606,82.854,372.848,-24.299,21.444,-41.938
C03163=1016.607,82.501,372.881,-24.299,21.444,-41.942
C03164=1016.608,82.148,372.915,-24.298,21.444,-41.945
C03165=1016.609,81.793,372.950,-24.298,21.445,-41.947
C03166=1016.611,81.438,372.984,-24.298,21.446,-41.951
C03167=1016.612,81.082,373.018,-24.297,21.445,-41.955
C03168=1016.613,80.725,373.052,-24.297,21.446,-41.958
C03169=1016.614,80.369,373.087,-24.296,21.446,-41.962
C03170=1016.615,80.014,373.121,-24.296,21.446,-41.964
C03171=1016.616,79.662,373.154,-24.295,21.447,-41.968
C03172=1016.617,79.318,373.187,-24.295,21.446,-41.971
C03173=1016.618,78.979,373.219,-24.295,21.448,-41.973
C03174=1016.619,78.646,373.251,-24.294,21.447,-41.977
C03175=1016.621,78.318,373.282,-24.293,21.448,-41.980
C03176=1016.622,77.994,373.314,-24.293,21.448,-41.984
C03177=1016.622,77.671,373.345,-24.292,21.448,-41.987
C03178=1016.624,77.346,373.376,-24.292,21.449,-41.990
C03179=1016.625,77.021,373.407,-24.292,21.449,-41.994
C03180=1016.626,76.690,373.439,-24.291,21.449,-41.997
C03181=1016.627,76.354,373.471,-24.291,21.449,-42.001
C03182=1016.628,76.012,373.504,-24.290,21.449,-42.004
C03183=1016.629,75.663,373.537,-24.290,21.450,-42.006
C03184=1016.631,75.309,373.571,-24.289,21.450,-42.010
C03185=1016.631,74.952,373.605,-24.289,21.450,-42.013
C03186=1016.633,74.594,373.639,-24.288,21.451,-42.017
C03187=1016.634,74.237,373.672,-24.288,21.451,-42.019
C03188=1016.634,73.882,373.706,-24.288,21.451,-42.023
C03189=1016.636,73.528,373.740,-24.287,21.452,-42.027
C03190=1016.637,73.177,373.773,-24.286,21.451,-42.030
C03191=1016.638,72.827,373.806,-24.286,21.452,-42.034
C03192=1016.640,72.479,373.840,-24.285,21.452,-42.037
C03193=1016.641,72.133,373.873,-24.285,21.453,-42.041
C03194=1016.641,71.787,373.906,-24.285,21.453,-42.043
C03195=1016.643,71.443,373.938,-24.284,21.453,-42.047
C03196=1016.643,71.098,373.971,-24.284,21.454,-42.051
C03197=1016.645,70.754,374.004,-24.283,21.453,-42.054
C03198=1016.646,70.409,374.036,-24.283,21.454,-42.058
C03199=1016.647,70.065,374.069,-24.282,21.454,-42.061
C03200=1016.648,69.720,374.102,-24.282,21.455,-42.063
C03201=1016.649,69.376,374.135,-24.281,21.455,-42.067
C03202=1016.649,69.033,374.167,-24.281,21.456,-42.071
C03203=1016.651,68.692,374.199,-24.280,21.455,-42.074
C03204=1016.652,68.350,374.231,-24.280,21.456,-42.078
C03205=1016.652,68.010,374.264,-24.279,21.456,-42.082
C03206=1016.654,67.670,374.295,-24.279,21.456,-42.085
C03207=1016.655,67.332,374.328,-24.279,21.457,-42.087
C03208=1016.656,66.995,374.359,-24.278,21.457,-42.091
C03209=1016.657,66.658,374.391,-24.278,21.457,-42.094
C03210=1016.658,66.322,374.422,-24.277,21.457,-42.098
C03211=1016.659,65.989,374.454,-24.277,21.458,-42.102
C03212=1016.660,65.650,374.486,-24.276,21.457,-42.105
C03213=1016.661,65.296,374.519,-24.276,21.459,-42.108
C03214=1016.662,64.919,374.555,-24.275,21.458,-42.113
C03215=1016.663,64.524,374.592,-24.274,21.459,-42.116
C03216=1016.664,64.137,374.628,-24.274,21.459,-42.120
C03217=1016.665,63.782,374.662,-24.274,21.460,-42.124
C03218=1016.667,63.408,374.696,-24.273,21.460,-42.128
C03219=1016.670,63.189,374.716,-24.273,21.461,-42.130
C03220=1016.673,62.966,374.734,-24.272,21.460,-42.131
C03221=1016.679,62.570,374.769,-24.272,21.460,-42.135
C03222=1016.684,62.234,374.798,-24.271,21.461,-42.139
C03223=1016.689,61.898,374.828,-24.271,21.461,-42.142
C03224=1016.693,61.563,374.856,-24.270,21.462,-42.146
C03225=1016.699,61.228,374.885,-24.270,21.461,-42.149
C03226=1016.703,60.894,374.915,-24.269,21.462,-42.153
C03227=1016.707,60.558,374.944,-24.269,21.462,-42.157
C03228=1016.712,60.224,374.973,-24.268,21.462,-42.160
C03229=1016.717,59.889,375.002,-24.268,21.463,-42.163
C03230=1016.722,59.554,375.030,-24.268,21.464,-42.166
C03231=1016.726,59.218,375.060,-24.267,21.464,-42.170
C03232=1016.731,58.883,375.088,-24.267,21.464,-42.173
C03233=1016.735,58.549,375.118,-24.266,21.464,-42.177
C03234=1016.740,58.214,375.147,-24.266,21.465,-42.181
C03235=1016.744,57.879,375.176,-24.265,21.464,-42.184
C03236=1016.750,57.544,375.205,-24.264,21.465,-42.188
C03237=1016.753,57.208,375.234,-24.264,21.465,-42.192
C03238=1016.758,56.874,375.262,-24.264,21.466,-42.194
C03239=1016.763,56.539,375.291,-24.263,21.466,-42.197
C03240=1016.767,56.204,375.321,-24.263,21.466,-42.201
C03241=1016.771,55.869,375.350,-24.262,21.467,-42.205
C03242=1016.775,55.534,375.378,-24.262,21.467,-42.209
C03243=1016.781,55.199,375.408,-24.261,21.467,-42.212
C03244=1016.785,54.864,375.436,-24.261,21.467,-42.216
C03245=1016.789,54.528,375.465,-24.260,21.468,-42.220
C03246=1016.793,54.194,375.494,-24.260,21.468,-42.223
C03247=1016.797,53.859,375.523,-24.259,21.468,-42.227
C03248=1016.802,53.524,375.552,-24.259,21.468,-42.230
C03249=1016.807,53.189,375.581,-24.258,21.469,-42.234
C03250=1016.811,52.854,375.610,-24.258,21.469,-42.238
C03251=1016.814,52.610,375.631,-24.257,21.470,-42.240
C03252=1016.818,52.275,375.660,-24.257,21.470,-42.244
C03253=1016.823,51.849,375.697,-24.256,21.470,-42.247
C03254=1016.827,51.514,375.725,-24.256,21.471,-42.251
C03255=1016.832,51.179,375.754,-24.255,21.471,-42.254
C03256=1016.836,50.844,375.783,-24.255,21.471,-42.258
C03257=1016.840,50.509,375.811,-24.254,21.471,-42.262
C03258=1016.844,50.174,375.840,-24.254,21.472,-42.266
C03259=1016.849,49.839,375.869,-24.253,21.472,-42.269
C03260=1016.852,49.504,375.898,-24.253,21.472,-42.273
C03261=1016.857,49.169,375.927,-24.252,21.473,-42.277
C03262=1016.861,48.834,375.956,-24.252,21.473,-42.280
C03263=1016.865,48.499,375.984,-24.251,21.473,-42.284
C03264=1016.869,48.164,376.013,-24.251,21.473,-42.287
C03265=1016.874,47.829,376.042,-24.250,21.474,-42.291
C03266=1016.877,47.494,376.072,-24.250,21.474,-42.295
C03267=1016.881,47.160,376.100,-24.249,21.475,-42.299
C03268=1016.885,46.825,376.128,-24.249,21.475,-42.302
C03269=1016.889,46.490,376.157,-24.248,21.475,-42.306
C03270=1016.893,46.154,376.186,-24.248,21.475,-42.309
C03271=1016.898,45.820,376.215,-24.247,21.476,-42.313
C03272=1016.901,45.485,376.243,-24.247,21.476,-42.317
C03273=1016.905,45.150,376.272,-24.246,21.477,-42.321
C03274=1016.909,44.815,376.301,-24.246,21.477,-42.325
C03275=1016.914,44.480,376.329,-24.245,21.477,-42.328
C03276=1016.917,44.146,376.358,-24.245,21.477,-42.332
C03277=1016.921,43.811,376.387,-24.244,21.478,-42.335
C03278=1016.925,43.476,376.416,-24.244,21.478,-42.339
C03279=1016.929,43.141,376.444,-24.243,21.479,-42.343
C03280=1016.933,42.806,376.473,-24.243,21.479,-42.347
C03281=1016.936,42.471,376.502,-24.242,21.479,-42.350
C03282=1016.940,42.137,376.530,-24.242,21.479,-42.354
C03283=1016.943,41.801,376.559,-24.241,21.480,-42.357
C03284=1016.948,41.467,376.587,-24.241,21.480,-42.361
C03285=1016.952,41.131,376.616,-24.240,21.481,-42.365
C03286=1016.955,40.798,376.645,-24.240,21.481,-42.369
C03287=1016.958,40.462,376.673,-24.239,21.481,-42.372
C03288=1016.963,40.128,376.702,-24.239,21.481,-42.376
C03289=1016.966,39.793,376.730,-24.238,21.482,-42.380
C03290=1016.970,39.459,376.759,-24.238,21.482,-42.383
C03291=1016.973,39.123,376.788,-24.237,21.483,-42.387
C03292=1016.977,38.788,376.816,-24.237,21.483,-42.391
C03293=1016.981,38.454,376.844,-24.236,21.483,-42.395
C03294=1016.984,38.119,376.873,-24.236,21.483,-42.398
C03295=1016.988,37.784,376.902,-24.235,21.484,-42.402
C03296=1016.992,37.449,376.930,-24.235,21.484,-42.405
C03297=1016.995,37.115,376.958,-24.234,21.485,-42.409
C03298=1016.998,36.780,376.987,-24.234,21.485,-42.413
C03299=1017.003,36.446,377.016,-24.233,21.485,-42.418
C03300=1017.006,36.110,377.044,-24.232,21.485,-42.422
C03301=1017.009,35.776,377.073,-24.232,21.486,-42.426
C03302=1017.013,35.442,377.101,-24.231,21.485,-42.429
C03303=1017.016,35.106,377.129,-24.231,21.486,-42.433
C03304=1017.020,34.772,377.157,-24.230,21.486,-42.437
C03305=1017.023,34.437,377.187,-24.230,21.487,-42.440
C03306=1017.027,34.103,377.215,-24.229,21.487,-42.444
C03307=1017.030,33.768,377.243,-24.229,21.488,-42.448
C03308=1017.034,33.434,377.272,-24.228,21.488,-42.452
C03309=1017.037,33.099,377.300,-24.228,21.489,-42.455
C03310=1017.041,32.764,377.328,-24.227,21.489,-42.459
C03311=1017.043,32.430,377.357,-24.226,21.489,-42.464
C03312=1017.047,32.096,377.385,-24.226,21.489,-42.468
C03313=1017.050,31.760,377.413,-24.225,21.489,-42.471
C03314=1017.054,31.427,377.442,-24.225,21.490,-42.475
C03315=1017.057,31.092,377.470,-24.224,21.490,-42.479
C03316=1017.060,30.757,377.498,-24.224,21.491,-42.483
C03317=1017.063,30.423,377.527,-24.223,21.491,-42.486
C03318=1017.067,30.089,377.555,-24.223,21.492,-42.490
C03319=1017.070,29.754,377.584,-24.222,21.492,-42.494
C03320=1017.073,29.420,377.612,-24.222,21.493,-42.498
C03321=1017.076,29.085,377.640,-24.221,21.492,-42.503
C03322=1017.079,28.751,377.668,-24.221,21.493,-42.507
C03323=1017.082,28.416,377.696,-24.220,21.493,-42.510
C03324=1017.086,28.082,377.725,-24.220,21.494,-42.514
C03325=1017.089,27.747,377.753,-24.219,21.494,-42.518
C03326=1017.092,27.413,377.781,-24.219,21.495,-42.522
C03327=1017.095,27.078,377.810,-24.218,21.494,-42.525
C03328=1017.098,26.744,377.837,-24.217,21.494,-42.530
C03329=1017.101,26.410,377.866,-24.217,21.495,-42.534
C03330=1017.105,26.076,377.894,-24.216,21.495,-42.538
C03331=1017.107,25.741,377.922,-24.216,21.496,-42.541
C03332=1017.110,25.407,377.951,-24.215,21.496,-42.545
C03333=1017.114,25.073,377.978,-24.215,21.497,-42.549
C03334=1017.116,24.738,378.007,-24.214,21.497,-42.553
C03335=1017.119,24.404,378.034,-24.213,21.497,-42.558
C03336=1017.122,24.078,378.062,-24.213,21.498,-42.560
C03337=1017.125,23.783,378.087,-24.213,21.498,-42.562
C03338=1017.127,23.531,378.108,-24.212,21.498,-42.565
C03339=1017.130,23.123,378.142,-24.211,21.499,-42.573
C03340=1017.134,22.714,378.177,-24.210,21.499,-42.580
C03341=1017.137,22.460,378.198,-24.210,21.500,-42.582
C03342=1017.139,22.167,378.223,-24.210,21.501,-42.584
C03343=1017.142,21.842,378.250,-24.209,21.500,-42.588
C03344=1017.144,21.486,378.280,-24.209,21.501,-42.593
C03345=1017.146,21.278,378.297,-24.208,21.501,-42.597
C03346=1017.149,21.052,378.316,-24.208,21.502,-42.599
C03347=1017.151,20.809,378.337,-24.208,21.502,-42.601
C03348=1017.152,20.562,378.358,-24.207,21.502,-42.603
C03349=1017.155,20.315,378.378,-24.207,21.502,-42.604
C03350=1017.157,20.079,378.399,-24.207,21.502,-42.608
C03351=1017.160,19.661,378.433,-24.206,21.503,-42.613
C03352=1017.163,19.313,378.462,-24.205,21.502,-42.619
C03353=1017.165,18.982,378.490,-24.205,21.503,-42.622
C03354=1017.168,18.649,378.518,-24.204,21.503,-42.626
C03355=1017.171,18.318,378.545,-24.204,21.504,-42.630
C03356=1017.174,17.987,378.573,-24.203,21.504,-42.634
C03357=1017.176,17.657,378.601,-24.202,21.504,-42.639
C03358=1017.179,17.327,378.628,-24.202,21.505,-42.643
C03359=1017.182,16.998,378.656,-24.201,21.505,-42.646
C03360=1017.184,16.670,378.683,-24.201,21.506,-42.650
C03361=1017.187,16.342,378.711,-24.200,21.506,-42.654
C03362=1017.189,16.014,378.738,-24.200,21.507,-42.658
C03363=1017.192,15.687,378.765,-24.199,21.507,-42.663
C03364=1017.195,15.360,378.792,-24.199,21.507,-42.667
C03365=1017.198,15.034,378.819,-24.198,21.508,-42.670
C03366=1017.200,14.709,378.847,-24.198,21.508,-42.674
C03367=1017.202,14.384,378.873,-24.197,21.509,-42.678
C03368=1017.205,14.059,378.901,-24.197,21.509,-42.682
C03369=1017.207,13.735,378.927,-24.196,21.509,-42.687
C03370=1017.210,13.411,378.954,-24.195,21.509,-42.691
C03371=1017.212,13.087,378.982,-24.195,21.510,-42.694
C03372=1017.214,12.763,379.008,-24.194,21.510,-42.698
C03373=1017.217,12.440,379.035,-24.194,21.511,-42.702
C03374=1017.219,12.116,379.062,-24.193,21.511,-42.707
C03375=1017.221,11.793,379.089,-24.193,21.511,-42.711
C03376=1017.224,11.470,379.115,-24.192,21.512,-42.715
C03377=1017.226,11.148,379.143,-24.192,21.512,-42.718
C03378=1017.228,10.827,379.169,-24.191,21.513,-42.722
C03379=1017.230,10.508,379.195,-24.191,21.513,-42.726
C03380=1017.233,10.191,379.222,-24.190,21.514,-42.730
C03381=1017.235,9.875,379.248,-24.190,21.514,-42.733
C03382=1017.237,9.561,379.274,-24.189,21.514,-42.738
C03383=1017.240,9.246,379.300,-24.188,21.515,-42.742
C03384=1017.241,8.931,379.326,-24.188,21.515,-42.746
C03385=1017.244,8.615,379.352,-24.187,21.516,-42.750
C03386=1017.246,8.296,379.378,-24.186,21.515,-42.755
C03387=1017.248,7.975,379.405,-24.186,21.516,-42.759
C03388=1017.250,7.653,379.432,-24.186,21.516,-42.762
C03389=1017.253,7.327,379.458,-24.185,21.517,-42.766
C03390=1017.255,7.000,379.486,-24.185,21.517,-42.770
C03391=1017.256,6.671,379.513,-24.184,21.518,-42.774
C03392=1017.259,6.342,379.540,-24.183,21.518,-42.779
C03393=1017.261,6.012,379.568,-24.183,21.518,-42.783
C03394=1017.263,5.683,379.594,-24.182,21.519,-42.786
C03395=1017.266,5.352,379.622,-24.181,21.518,-42.792
C03396=1017.268,5.021,379.649,-24.181,21.519,-42.795
C03397=1017.270,4.691,379.676,-24.180,21.519,-42.799
C03398=1017.272,4.359,379.703,-24.180,21.521,-42.803
C03399=1017.274,4.030,379.730,-24.179,21.520,-42.807
C03400=1017.276,3.716,379.756,-24.179,21.521,-42.810
C03401=1017.278,3.427,379.780,-24.179,21.521,-42.814
C03402=1017.279,3.157,379.802,-24.178,21.522,-42.818
C03403=1017.281,2.895,379.824,-24.177,21.522,-42.823
C03404=1017.282,2.627,379.846,-24.177,21.522,-42.827
C03405=1017.284,2.338,379.869,-24.176,21.523,-42.831
C03406=1017.286,2.026,379.895,-24.176,21.523,-42.834
C03407=1017.289,1.695,379.922,-24.175,21.523,-42.838
C03408=1017.291,1.362,379.949,-24.175,21.524,-42.842
C03409=1017.292,1.028,379.977,-24.174,21.525,-42.846
C03410=1017.294,0.693,380.004,-24.173,21.525,-42.851
C03411=1017.296,0.358,380.032,-24.173,21.525,-42.855
C03412=1017.298,0.020,380.059,-24.172,21.526,-42.858
C03413=1017.300,-0.318,380.087,-24.172,21.526,-42.864
C03414=1017.302,-0.658,380.115,-24.171,21.526,-42.867
C03415=1017.304,-1.001,380.143,-24.170,21.527,-42.873
C03416=1017.305,-1.343,380.171,-24.170,21.527,-42.877
C03417=1017.307,-1.689,380.199,-24.169,21.528,-42.880
C03418=1017.309,-2.036,380.227,-24.169,21.528,-42.886
C03419=1017.311,-2.383,380.256,-24.168,21.529,-42.890
C03420=1017.313,-2.733,380.284,-24.167,21.529,-42.895
C03421=1017.315,-3.085,380.313,-24.167,21.529,-42.899
C03422=1017.317,-3.437,380.342,-24.166,21.529,-42.904
C03423=1017.319,-3.792,380.371,-24.166,21.531,-42.908
C03424=1017.320,-4.149,380.400,-24.165,21.530,-42.913
C03425=1017.322,-4.511,380.429,-24.164,21.531,-42.919
C03426=1017.325,-4.877,380.459,-24.164,21.532,-42.923
C03427=1017.326,-5.247,380.489,-24.163,21.532,-42.928
C03428=1017.328,-5.621,380.520,-24.163,21.533,-42.932
C03429=1017.330,-5.996,380.551,-24.162,21.533,-42.937
C03430=1017.332,-6.371,380.581,-24.161,21.533,-42.941
C03431=1017.333,-6.746,380.611,-24.160,21.534,-42.947
C03432=1017.336,-7.117,380.641,-24.160,21.534,-42.952
C03433=1017.337,-7.487,380.671,-24.159,21.535,-42.956
C03434=1017.339,-7.853,380.700,-24.158,21.535,-42.961
C03435=1017.341,-8.216,380.731,-24.158,21.536,-42.967
C03436=1017.342,-8.579,380.760,-24.157,21.536,-42.971
C03437=1017.343,-8.942,380.789,-24.156,21.536,-42.976
C03438=1017.345,-9.304,380.818,-24.156,21.537,-42.982
C03439=1017.347,-9.666,380.847,-24.155,21.538,-42.985
C03440=1017.349,-10.028,380.876,-24.154,21.538,-42.991
C03441=1017.350,-10.389,380.906,-24.154,21.539,-42.995
C03442=1017.352,-10.749,380.936,-24.153,21.539,-43.000
C03443=1017.353,-11.108,380.964,-24.152,21.539,-43.006
C03444=1017.355,-11.466,380.992,-24.152,21.540,-43.009
C03445=1017.356,-11.821,381.021,-24.151,21.540,-43.014
C03446=1017.357,-12.177,381.050,-24.151,21.541,-43.019
C03447=1017.359,-12.531,381.078,-24.150,21.541,-43.024
C03448=1017.361,-12.883,381.107,-24.149,21.542,-43.028
C03449=1017.362,-13.233,381.135,-24.149,21.542,-43.033
C03450=1017.364,-13.581,381.163,-24.148,21.543,-43.037
C03451=1017.365,-13.928,381.191,-24.147,21.543,-43.042
C03452=1017.366,-14.271,381.219,-24.147,21.544,-43.046
C03453=1017.368,-14.614,381.246,-24.146,21.544,-43.052
C03454=1017.369,-14.953,381.273,-24.146,21.544,-43.055
C03455=1017.370,-15.292,381.301,-24.145,21.545,-43.061
C03456=1017.371,-15.628,381.328,-24.145,21.546,-43.065
C03457=1017.373,-15.963,381.354,-24.144,21.546,-43.070
C03458=1017.374,-16.298,381.381,-24.143,21.546,-43.074
C03459=1017.375,-16.631,381.408,-24.142,21.547,-43.079
C03460=1017.376,-16.965,381.434,-24.142,21.547,-43.083
C03461=1017.378,-17.297,381.461,-24.141,21.547,-43.088
C03462=1017.379,-17.630,381.488,-24.141,21.548,-43.092
C03463=1017.380,-17.996,381.517,-24.140,21.549,-43.100
C03464=1017.381,-18.217,381.535,-24.139,21.548,-43.103
C03465=1017.381,-18.465,381.554,-24.139,21.549,-43.105
C03466=1017.383,-18.726,381.576,-24.139,21.550,-43.107
C03467=1017.383,-18.989,381.597,-24.139,21.550,-43.109
C03468=1017.384,-19.236,381.616,-24.138,21.550,-43.112
C03469=1017.385,-19.653,381.650,-24.137,21.550,-43.118
C03470=1017.386,-19.825,381.663,-24.137,21.551,-43.122
C03471=1017.387,-20.158,381.690,-24.136,21.551,-43.127
C03472=1017.388,-20.490,381.716,-24.136,21.552,-43.131
C03473=1017.389,-20.823,381.743,-24.135,21.553,-43.135
C03474=1017.390,-21.156,381.770,-24.134,21.552,-43.140
C03475=1017.391,-21.489,381.795,-24.134,21.553,-43.144
C03476=1017.392,-21.822,381.822,-24.133,21.554,-43.149
C03477=1017.392,-22.154,381.848,-24.133,21.554,-43.153
C03478=1017.394,-22.487,381.875,-24.132,21.554,-43.158
C03479=1017.394,-22.820,381.901,-24.131,21.556,-43.162
C03480=1017.396,-23.153,381.928,-24.131,21.555,-43.168
C03481=1017.396,-23.486,381.954,-24.130,21.556,-43.171
C03482=1017.398,-23.818,381.981,-24.129,21.556,-43.177
C03483=1017.398,-24.151,382.007,-24.129,21.557,-43.181
C03484=1017.399,-24.484,382.034,-24.128,21.557,-43.186
C03485=1017.400,-24.817,382.060,-24.128,21.558,-43.190
C03486=1017.401,-25.149,382.086,-24.127,21.558,-43.195
C03487=1017.402,-25.482,382.113,-24.126,21.559,-43.199
C03488=1017.402,-25.815,382.139,-24.126,21.559,-43.204
C03489=1017.403,-26.148,382.165,-24.125,21.559,-43.208
C03490=1017.404,-26.481,382.191,-24.124,21.560,-43.214
C03491=1017.405,-26.813,382.218,-24.124,21.560,-43.217
C03492=1017.405,-27.146,382.244,-24.123,21.560,-43.223
C03493=1017.406,-27.479,382.270,-24.123,21.562,-43.227
C03494=1017.407,-27.811,382.296,-24.122,21.562,-43.232
C03495=1017.408,-28.144,382.323,-24.121,21.562,-43.236
C03496=1017.409,-28.477,382.349,-24.120,21.562,-43.241
C03497=1017.409,-28.810,382.375,-24.120,21.563,-43.245
C03498=1017.410,-29.142,382.401,-24.119,21.563,-43.250
C03499=1017.410,-29.476,382.428,-24.119,21.564,-43.254
C03500=1017.410,-29.808,382.454,-24.118,21.565,-43.260
C03501=1017.411,-30.141,382.479,-24.118,21.565,-43.264
C03502=1017.412,-30.474,382.506,-24.117,21.565,-43.269
C03503=1017.412,-30.806,382.532,-24.116,21.566,-43.273
C03504=1017.413,-31.139,382.558,-24.116,21.566,-43.278
C03505=1017.413,-31.472,382.584,-24.115,21.567,-43.282
C03506=1017.414,-31.804,382.610,-24.114,21.567,-43.287
C03507=1017.415,-32.137,382.636,-24.114,21.568,-43.291
C03508=1017.415,-32.470,382.662,-24.113,21.568,-43.296
C03509=1017.416,-32.803,382.688,-24.113,21.569,-43.301
C03510=1017.416,-33.135,382.714,-24.112,21.569,-43.306
C03511=1017.417,-33.468,382.741,-24.111,21.570,-43.310
C03512=1017.418,-33.801,382.766,-24.111,21.570,-43.315
C03513=1017.418,-34.133,382.793,-24.110,21.571,-43.319
C03514=1017.418,-34.465,382.818,-24.109,21.571,-43.324
C03515=1017.418,-34.799,382.844,-24.109,21.572,-43.328
C03516=1017.419,-35.132,382.871,-24.108,21.572,-43.334
C03517=1017.419,-35.464,382.897,-24.108,21.573,-43.337
C03518=1017.419,-35.797,382.922,-24.107,21.573,-43.343
C03519=1017.420,-36.130,382.948,-24.107,21.574,-43.347
C03520=1017.420,-36.462,382.974,-24.106,21.574,-43.352
C03521=1017.420,-36.795,382.999,-24.105,21.574,-43.357
C03522=1017.421,-37.128,383.026,-24.105,21.575,-43.361
C03523=1017.421,-37.460,383.052,-24.104,21.575,-43.366
C03524=1017.421,-37.793,383.077,-24.103,21.576,-43.371
C03525=1017.422,-38.125,383.103,-24.102,21.576,-43.376
C03526=1017.422,-38.458,383.129,-24.102,21.577,-43.380
C03527=1017.422,-38.791,383.155,-24.101,21.577,-43.385
C03528=1017.422,-39.124,383.181,-24.101,21.578,-43.389
C03529=1017.422,-39.456,383.207,-24.100,21.578,-43.394
C03530=1017.423,-39.789,383.232,-24.100,21.579,-43.398
C03531=1017.423,-40.122,383.258,-24.099,21.579,-43.404
C03532=1017.423,-40.454,383.284,-24.098,21.580,-43.409
C03533=1017.423,-40.787,383.309,-24.098,21.580,-43.413
C03534=1017.423,-41.119,383.335,-24.097,21.580,-43.418
C03535=1017.424,-41.452,383.361,-24.096,21.582,-43.422
C03536=1017.424,-41.784,383.386,-24.096,21.582,-43.427
C03537=1017.424,-42.117,383.412,-24.095,21.582,-43.431
C03538=1017.424,-42.449,383.438,-24.094,21.583,-43.437
C03539=1017.424,-42.783,383.464,-24.094,21.583,-43.442
C03540=1017.423,-43.115,383.489,-24.093,21.583,-43.446
C03541=1017.424,-43.448,383.515,-24.092,21.584,-43.451
C03542=1017.424,-43.780,383.540,-24.092,21.585,-43.455
C03543=1017.424,-44.112,383.566,-24.091,21.585,-43.461
C03544=1017.424,-44.445,383.591,-24.091,21.586,-43.465
C03545=1017.424,-44.777,383.617,-24.090,21.586,-43.470
C03546=1017.424,-45.110,383.643,-24.089,21.586,-43.475
C03547=1017.424,-45.443,383.668,-24.089,21.587,-43.479
C03548=1017.424,-45.775,383.694,-24.088,21.588,-43.485
C03549=1017.424,-46.107,383.719,-24.088,21.588,-43.488
C03550=1017.423,-46.441,383.745,-24.087,21.588,-43.494
C03551=1017.423,-46.773,383.770,-24.086,21.590,-43.498
C03552=1017.423,-47.106,383.795,-24.086,21.589,-43.503
C03553=1017.423,-47.438,383.821,-24.085,21.589,-43.508
C03554=1017.423,-47.770,383.847,-24.084,21.591,-43.512
C03555=1017.423,-48.103,383.872,-24.083,21.591,-43.518
C03556=1017.422,-48.435,383.897,-24.083,21.592,-43.522
C03557=1017.422,-48.767,383.923,-24.082,21.592,-43.527
C03558=1017.422,-49.100,383.948,-24.081,21.592,-43.532
C03559=1017.422,-49.432,383.974,-24.081,21.593,-43.536
C03560=1017.422,-49.765,383.999,-24.080,21.593,-43.542
C03561=1017.421,-50.097,384.024,-24.080,21.595,-43.546
C03562=1017.421,-50.429,384.050,-24.079,21.594,-43.551
C03563=1017.421,-50.762,384.075,-24.079,21.595,-43.555
C03564=1017.421,-51.094,384.100,-24.078,21.596,-43.560
C03565=1017.420,-51.426,384.125,-24.077,21.596,-43.566
C03566=1017.420,-51.759,384.150,-24.077,21.597,-43.570
C03567=1017.420,-52.091,384.176,-24.076,21.597,-43.575
C03568=1017.419,-52.423,384.201,-24.075,21.597,-43.579
C03569=1017.419,-52.756,384.226,-24.075,21.598,-43.584
C03570=1017.418,-53.088,384.252,-24.074,21.598,-43.589
C03571=1017.418,-53.420,384.277,-24.074,21.600,-43.594
C03572=1017.418,-53.753,384.302,-24.073,21.599,-43.599
C03573=1017.417,-54.085,384.327,-24.072,21.600,-43.603
C03574=1017.416,-54.417,384.353,-24.072,21.601,-43.608
C03575=1017.415,-54.750,384.377,-24.071,21.601,-43.613
C03576=1017.415,-55.082,384.403,-24.070,21.602,-43.618
C03577=1017.415,-55.415,384.428,-24.070,21.602,-43.623
C03578=1017.414,-55.747,384.453,-24.069,21.603,-43.627
C03579=1017.413,-56.081,384.478,-24.068,21.603,-43.632
C03580=1017.413,-56.413,384.503,-24.068,21.603,-43.637
C03581=1017.412,-56.747,384.528,-24.067,21.605,-43.642
C03582=1017.412,-57.080,384.554,-24.066,21.604,-43.647
C03583=1017.411,-57.414,384.579,-24.066,21.605,-43.652
C03584=1017.411,-57.747,384.604,-24.065,21.606,-43.656
C03585=1017.410,-58.082,384.629,-24.064,21.606,-43.662
C03586=1017.410,-58.416,384.654,-24.064,21.607,-43.666
C03587=1017.409,-58.751,384.679,-24.063,21.607,-43.671
C03588=1017.408,-59.087,384.704,-24.062,21.608,-43.676
C03589=1017.407,-59.422,384.730,-24.062,21.608,-43.680
C03590=1017.406,-59.758,384.754,-24.061,21.609,-43.686
C03591=1017.406,-60.094,384.780,-24.060,21.609,-43.691
C03592=1017.405,-60.431,384.806,-24.060,21.610,-43.695
C03593=1017.405,-60.768,384.830,-24.059,21.610,-43.700
C03594=1017.404,-61.106,384.856,-24.059,21.611,-43.706
C03595=1017.402,-61.444,384.881,-24.058,21.611,-43.710
C03596=1017.401,-61.783,384.907,-24.057,21.612,-43.715
C03597=1017.401,-62.121,384.932,-24.057,21.612,-43.720
C03598=1017.400,-62.461,384.957,-24.056,21.614,-43.725
C03599=1017.399,-62.800,384.983,-24.055,21.613,-43.730
C03600=1017.398,-63.140,385.008,-24.055,21.614,-43.735
C03601=1017.398,-63.480,385.034,-24.054,21.615,-43.739
C03602=1017.397,-63.821,385.059,-24.053,21.616,-43.745
C03603=1017.396,-64.162,385.085,-24.053,21.615,-43.750
C03604=1017.395,-64.504,385.110,-24.052,21.617,-43.754
C03605=1017.393,-64.845,385.135,-24.051,21.617,-43.759
C03606=1017.393,-65.187,385.161,-24.051,21.618,-43.765
C03607=1017.392,-65.529,385.186,-24.050,21.617,-43.770
C03608=1017.390,-65.871,385.211,-24.050,21.619,-43.774
C03609=1017.389,-66.214,385.237,-24.049,21.619,-43.780
C03610=1017.389,-66.557,385.263,-24.048,21.620,-43.785
C03611=1017.387,-66.900,385.288,-24.048,21.620,-43.789
C03612=1017.386,-67.242,385.314,-24.047,21.621,-43.795
C03613=1017.385,-67.586,385.339,-24.046,21.621,-43.800
C03614=1017.384,-67.929,385.364,-24.045,21.622,-43.805
C03615=1017.382,-68.273,385.390,-24.045,21.622,-43.809
C03616=1017.382,-68.616,385.415,-24.044,21.623,-43.815
C03617=1017.381,-68.961,385.440,-24.043,21.623,-43.820
C03618=1017.380,-69.305,385.466,-24.043,21.624,-43.824
C03619=1017.378,-69.649,385.491,-24.042,21.624,-43.829
C03620=1017.376,-69.993,385.517,-24.041,21.625,-43.835
C03621=1017.375,-70.337,385.542,-24.041,21.625,-43.840
C03622=1017.374,-70.681,385.568,-24.040,21.626,-43.844
C03623=1017.373,-71.025,385.594,-24.040,21.627,-43.850
C03624=1017.371,-71.369,385.618,-24.039,21.627,-43.855
C03625=1017.371,-71.713,385.644,-24.038,21.628,-43.861
C03626=1017.369,-72.056,385.669,-24.038,21.628,-43.865
C03627=1017.368,-72.401,385.694,-24.037,21.629,-43.870
C03628=1017.366,-72.745,385.720,-24.036,21.629,-43.875
C03629=1017.365,-73.089,385.745,-24.035,21.630,-43.881
C03630=1017.363,-73.433,385.770,-24.035,21.630,-43.885
C03631=1017.362,-73.777,385.796,-24.034,21.631,-43.890
C03632=1017.360,-74.120,385.821,-24.033,21.632,-43.896
C03633=1017.359,-74.463,385.846,-24.033,21.632,-43.901
C03634=1017.358,-74.807,385.871,-24.032,21.633,-43.905
C03635=1017.356,-75.150,385.896,-24.031,21.633,-43.911
C03636=1017.354,-75.494,385.921,-24.031,21.634,-43.916
C03637=1017.353,-75.837,385.946,-24.030,21.634,-43.920
C03638=1017.351,-76.180,385.971,-24.030,21.635,-43.926
C03639=1017.350,-76.522,385.996,-24.029,21.635,-43.931
C03640=1017.348,-76.865,386.021,-24.028,21.636,-43.936
C03641=1017.347,-77.207,386.047,-24.028,21.636,-43.940
C03642=1017.346,-77.549,386.072,-24.027,21.637,-43.946
C03643=1017.343,-77.891,386.096,-24.026,21.637,-43.951
C03644=1017.341,-78.232,386.121,-24.026,21.639,-43.955
C03645=1017.340,-78.574,386.147,-24.025,21.638,-43.960
C03646=1017.339,-78.914,386.171,-24.024,21.639,-43.966
C03647=1017.337,-79.255,386.196,-24.023,21.639,-43.971
